// Mitsubishi GX Works2 project: LG WM Press 21.07.21_Conv   PLC: Q03UDV
// LG WM Press 21.07.21_Conv

PROGRAM MAIN
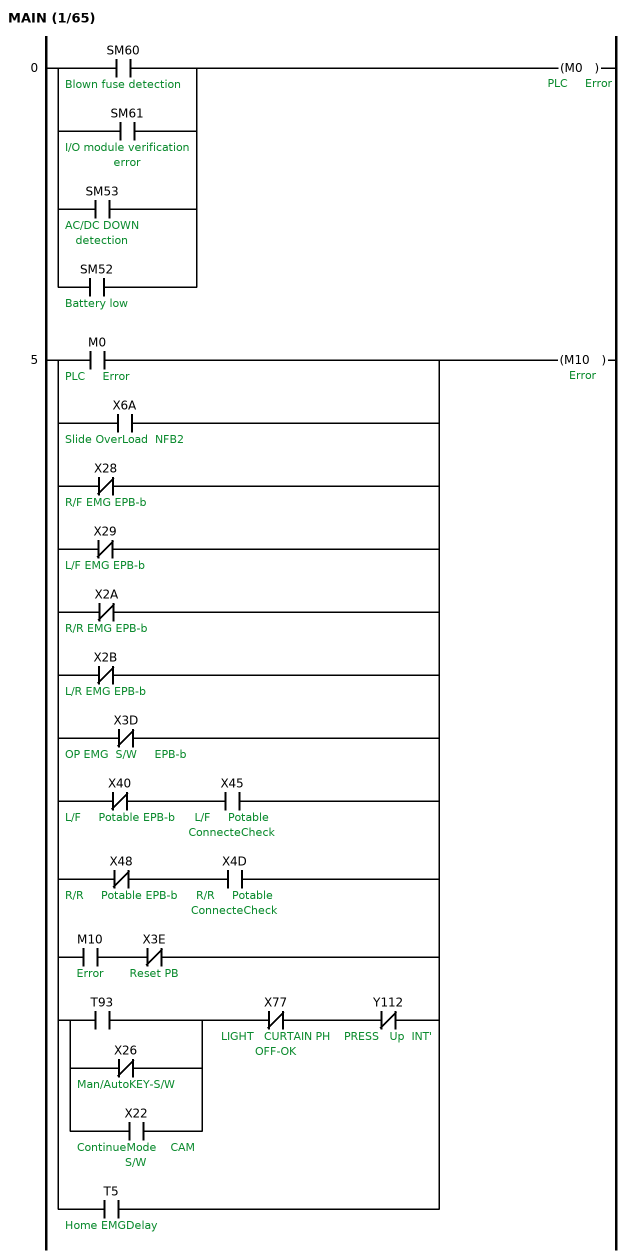
0     LD      SM60  ; Blown fuse detection
      OR      SM61  ; I/O module verification error
      OR      SM53  ; AC/DC DOWN detection
      OR      SM52  ; Battery low
      OUT     M0  ; PLC     Error
5     LD      M0  ; PLC     Error
      OR      X6A  ; Slide OverLoad  NFB2
      ORI     X28  ; R/F EMG EPB-b
      ORI     X29  ; L/F EMG EPB-b
      ORI     X2A  ; R/R EMG EPB-b
      ORI     X2B  ; L/R EMG EPB-b
      ORI     X3D  ; OP EMG  S/W     EPB-b
      LDI     X40  ; L/F     Potable EPB-b
      AND     X45  ; L/F     Potable ConnecteCheck
      ORB
      LDI     X48  ; R/R     Potable EPB-b
      AND     X4D  ; R/R     Potable ConnecteCheck
      ORB
      LD      M10  ; Error
      ANI     X3E  ; Reset PB
      ORB
      LD      T93
      ORI     X26  ; Man/AutoKEY-S/W
      OR      X22  ; ContinueMode    CAM S/W
      ANI     X77  ; LIGHT   CURTAIN PH      OFF-OK
      ANI     Y112  ; PRESS   Up  INT'
      ORB
      OR      T5  ; Home EMGDelay
      OUT     M10  ; Error
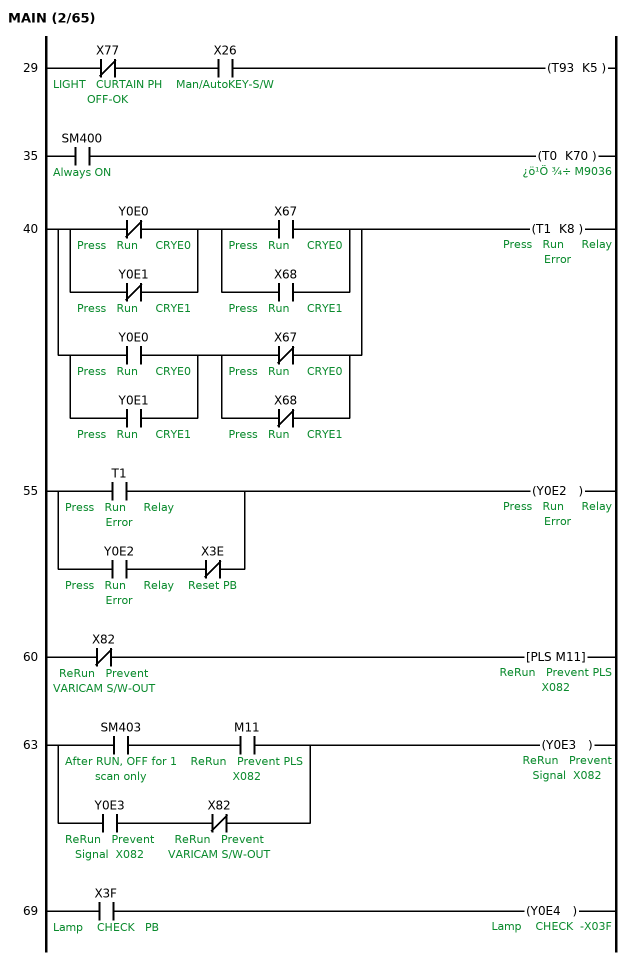
29    LDI     X77  ; LIGHT   CURTAIN PH      OFF-OK
      AND     X26  ; Man/AutoKEY-S/W
      OUT     T93 K5
35    LD      SM400  ; Always ON
      OUT     T0 K70  ; ¿ö¹Ö ¾÷ M9036
40    LDI     Y0E0  ; Press   Run     CRYE0
      ORI     Y0E1  ; Press   Run     CRYE1
      LD      X67  ; Press   Run     CRYE0
      OR      X68  ; Press   Run     CRYE1
      ANB
      LD      Y0E0  ; Press   Run     CRYE0
      OR      Y0E1  ; Press   Run     CRYE1
      LDI     X67  ; Press   Run     CRYE0
      ORI     X68  ; Press   Run     CRYE1
      ANB
      ORB
      OUT     T1 K8  ; Press   Run     Relay   Error
55    LD      T1  ; Press   Run     Relay   Error
      LD      Y0E2  ; Press   Run     Relay   Error
      ANI     X3E  ; Reset PB
      ORB
      OUT     Y0E2  ; Press   Run     Relay   Error
60    LDI     X82  ; ReRun   Prevent VARICAM S/W-OUT
      PLS     M11  ; ReRun   Prevent PLS X082
63    LD      SM403  ; After RUN, OFF for 1 scan only
      AND     M11  ; ReRun   Prevent PLS X082
      LD      Y0E3  ; ReRun   Prevent Signal  X082
      ANI     X82  ; ReRun   Prevent VARICAM S/W-OUT
      ORB
      OUT     Y0E3  ; ReRun   Prevent Signal  X082
69    LD      X3F  ; Lamp    CHECK   PB
      OUT     Y0E4  ; Lamp    CHECK  -X03F
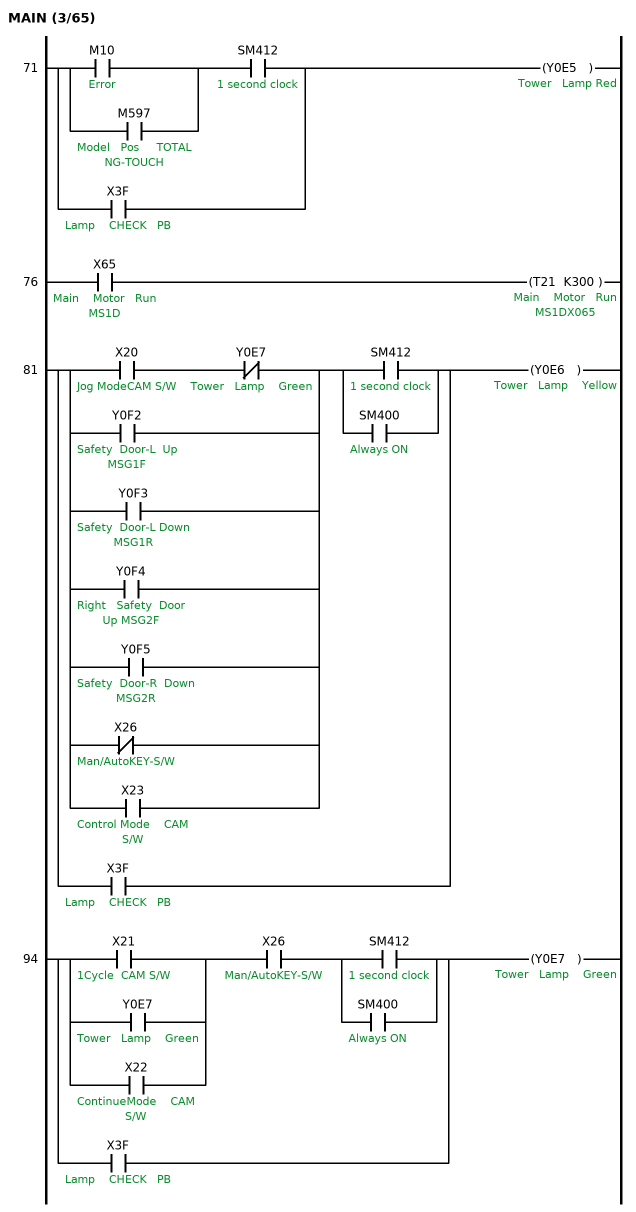
71    LD      M10  ; Error
      OR      M597  ; Model   Pos     TOTAL   NG-TOUCH
      AND     SM412  ; 1 second clock
      OR      X3F  ; Lamp    CHECK   PB
      OUT     Y0E5  ; Tower   Lamp Red
76    LD      X65  ; Main    Motor   Run MS1D
      OUT     T21 K300  ; Main    Motor   Run MS1DX065
81    LD      X20  ; Jog ModeCAM S/W
      ANI     Y0E7  ; Tower   Lamp    Green
      OR      Y0F2  ; Safety  Door-L  Up MSG1F
      OR      Y0F3  ; Safety  Door-L Down     MSG1R
      OR      Y0F4  ; Right   Safety  Door Up MSG2F
      OR      Y0F5  ; Safety  Door-R  Down    MSG2R
      ORI     X26  ; Man/AutoKEY-S/W
      OR      X23  ; Control Mode    CAM S/W
      LD      SM412  ; 1 second clock
      OR      SM400  ; Always ON
      ANB
      OR      X3F  ; Lamp    CHECK   PB
      OUT     Y0E6  ; Tower   Lamp    Yellow
94    LD      X21  ; 1Cycle  CAM S/W
      OR      Y0E7  ; Tower   Lamp    Green
      OR      X22  ; ContinueMode    CAM S/W
      AND     X26  ; Man/AutoKEY-S/W
      LD      SM412  ; 1 second clock
      OR      SM400  ; Always ON
      ANB
      OR      X3F  ; Lamp    CHECK   PB
      OUT     Y0E7  ; Tower   Lamp    Green
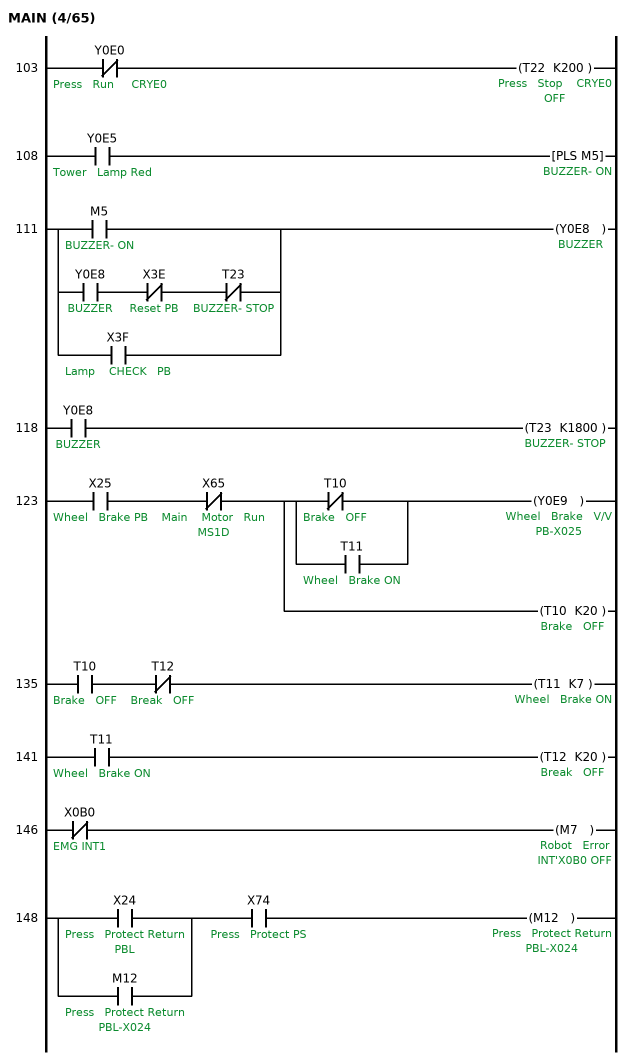
103   LDI     Y0E0  ; Press   Run     CRYE0
      OUT     T22 K200  ; Press   Stop    CRYE0   OFF
108   LD      Y0E5  ; Tower   Lamp Red
      PLS     M5  ; BUZZER- ON
111   LD      M5  ; BUZZER- ON
      LD      Y0E8  ; BUZZER
      ANI     X3E  ; Reset PB
      ANI     T23  ; BUZZER- STOP
      ORB
      OR      X3F  ; Lamp    CHECK   PB
      OUT     Y0E8  ; BUZZER
118   LD      Y0E8  ; BUZZER
      OUT     T23 K1800  ; BUZZER- STOP
123   LD      X25  ; Wheel   Brake PB
      ANI     X65  ; Main    Motor   Run MS1D
      MPS
      LDI     T10  ; Brake   OFF
      OR      T11  ; Wheel   Brake ON
      ANB
      OUT     Y0E9  ; Wheel   Brake   V/V     PB-X025
      MPP
      OUT     T10 K20  ; Brake   OFF
135   LD      T10  ; Brake   OFF
      ANI     T12  ; Break   OFF
      OUT     T11 K7  ; Wheel   Brake ON
141   LD      T11  ; Wheel   Brake ON
      OUT     T12 K20  ; Break   OFF
146   LDI     X0B0  ; EMG INT1
      OUT     M7  ; Robot   Error   INT'X0B0 OFF
148   LD      X24  ; Press   Protect Return  PBL
      OR      M12  ; Press   Protect Return  PBL-X024
      AND     X74  ; Press   Protect PS
      OUT     M12  ; Press   Protect Return  PBL-X024
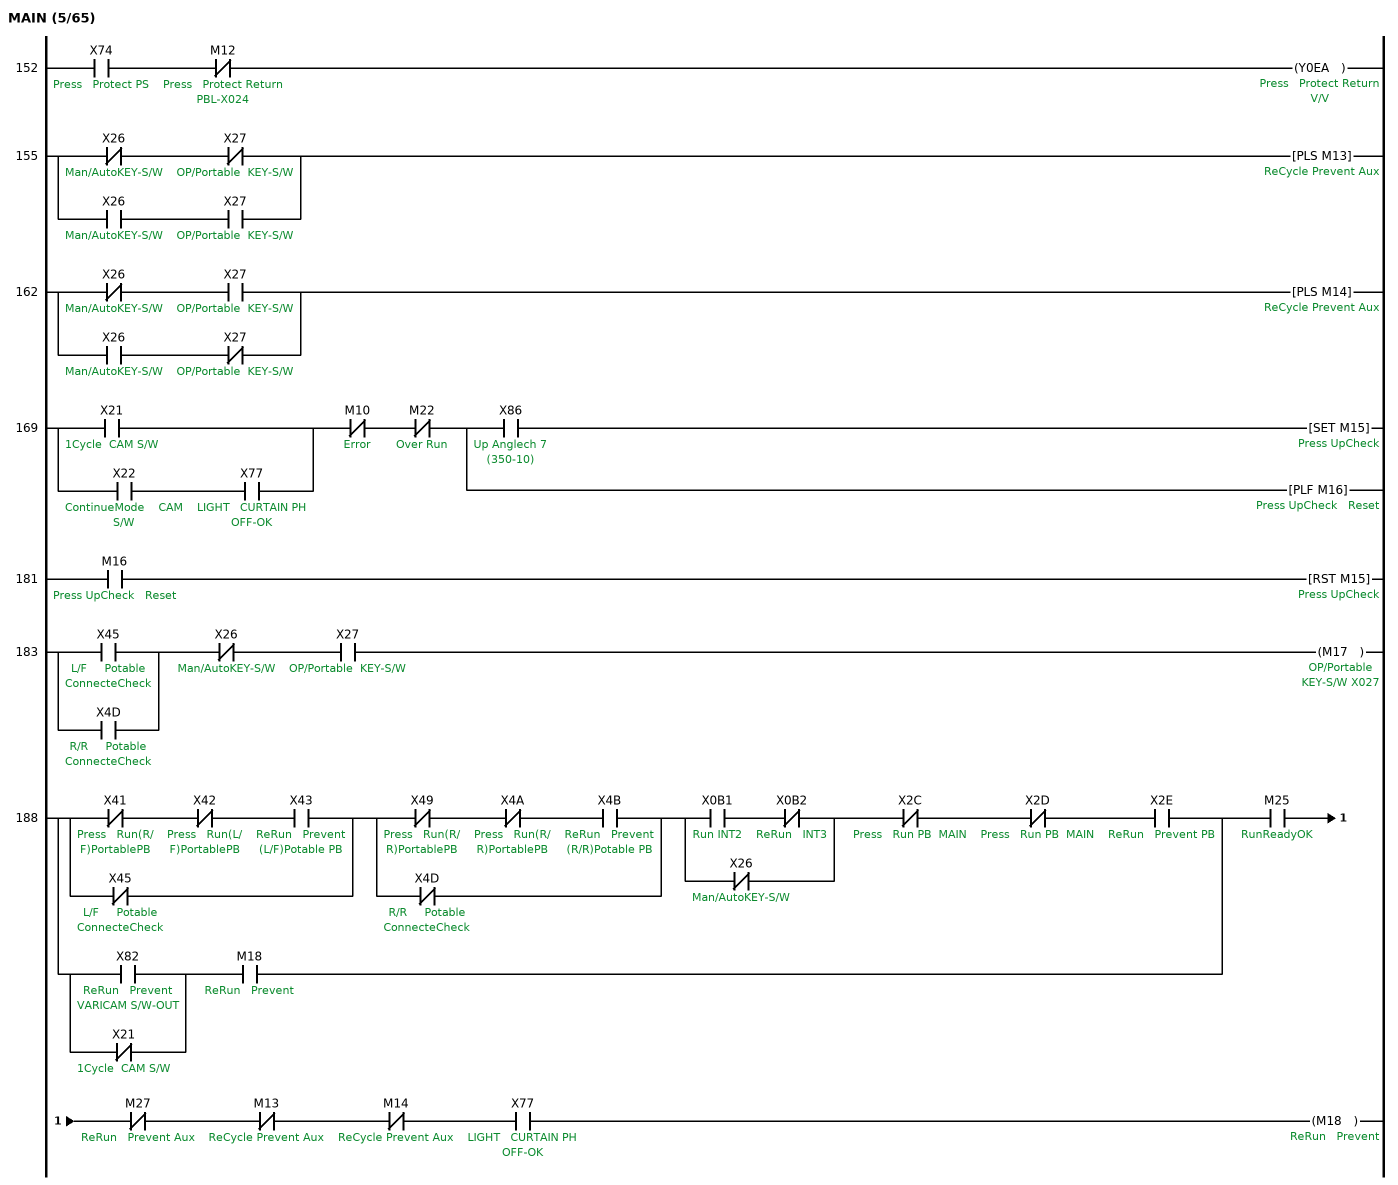
152   LD      X74  ; Press   Protect PS
      ANI     M12  ; Press   Protect Return  PBL-X024
      OUT     Y0EA  ; Press   Protect Return  V/V
155   LDI     X26  ; Man/AutoKEY-S/W
      ANI     X27  ; OP/Portable  KEY-S/W
      LD      X26  ; Man/AutoKEY-S/W
      AND     X27  ; OP/Portable  KEY-S/W
      ORB
      PLS     M13  ; ReCycle Prevent Aux
162   LDI     X26  ; Man/AutoKEY-S/W
      AND     X27  ; OP/Portable  KEY-S/W
      LD      X26  ; Man/AutoKEY-S/W
      ANI     X27  ; OP/Portable  KEY-S/W
      ORB
      PLS     M14  ; ReCycle Prevent Aux
169   LD      X21  ; 1Cycle  CAM S/W
      LD      X22  ; ContinueMode    CAM S/W
      AND     X77  ; LIGHT   CURTAIN PH      OFF-OK
      ORB
      ANI     M10  ; Error
      ANI     M22  ; Over Run
      MPS
      AND     X86  ; Up Anglech 7    (350-10)
      SET     M15  ; Press UpCheck
      MPP
      PLF     M16  ; Press UpCheck   Reset
181   LD      M16  ; Press UpCheck   Reset
      RST     M15  ; Press UpCheck
183   LD      X45  ; L/F     Potable ConnecteCheck
      OR      X4D  ; R/R     Potable ConnecteCheck
      ANI     X26  ; Man/AutoKEY-S/W
      AND     X27  ; OP/Portable  KEY-S/W
      OUT     M17  ; OP/Portable     KEY-S/W X027
188   LDI     X41  ; Press   Run(R/F)PortablePB
      ANI     X42  ; Press   Run(L/F)PortablePB
      AND     X43  ; ReRun   Prevent (L/F)Potable PB
      ORI     X45  ; L/F     Potable ConnecteCheck
      LDI     X49  ; Press   Run(R/R)PortablePB
      ANI     X4A  ; Press   Run(R/R)PortablePB
      AND     X4B  ; ReRun   Prevent (R/R)Potable PB
      ORI     X4D  ; R/R     Potable ConnecteCheck
      ANB
      LD      X0B1  ; Run INT2
      ANI     X0B2  ; ReRun   INT3
      ORI     X26  ; Man/AutoKEY-S/W
      ANB
      ANI     X2C  ; Press   Run PB  MAIN
      ANI     X2D  ; Press   Run PB  MAIN
      AND     X2E  ; ReRun   Prevent PB
      LD      X82  ; ReRun   Prevent VARICAM S/W-OUT
      ORI     X21  ; 1Cycle  CAM S/W
      AND     M18  ; ReRun   Prevent
      ORB
      AND     M25  ; RunReadyOK
      ANI     M27  ; ReRun   Prevent Aux
      ANI     M13  ; ReCycle Prevent Aux
      ANI     M14  ; ReCycle Prevent Aux
      AND     X77  ; LIGHT   CURTAIN PH      OFF-OK
      OUT     M18  ; ReRun   Prevent
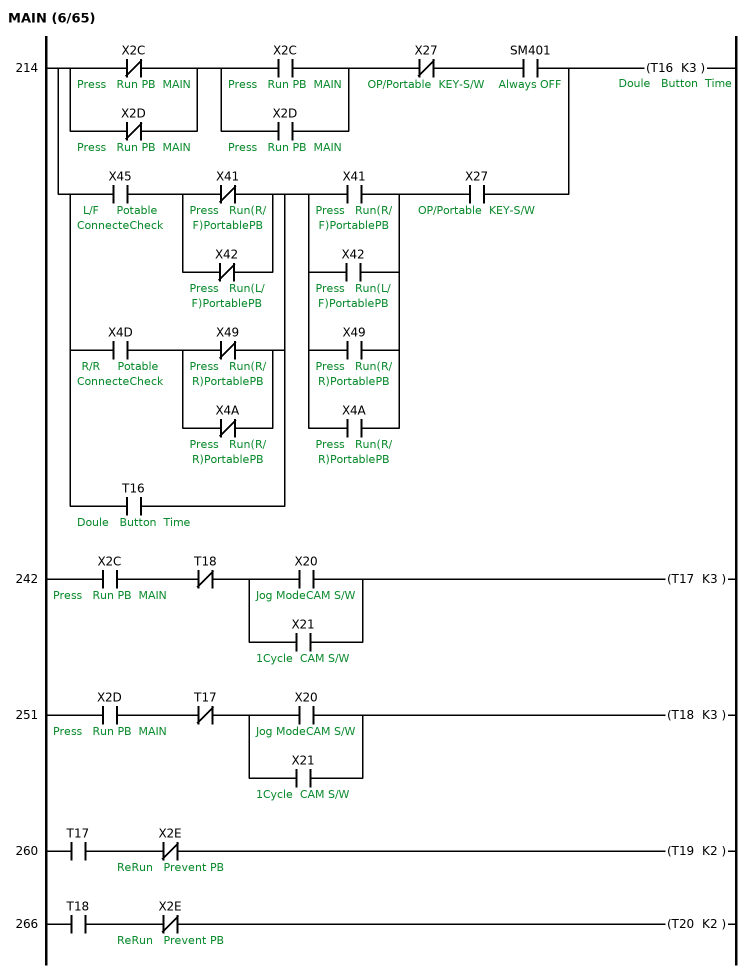
214   LDI     X2C  ; Press   Run PB  MAIN
      ORI     X2D  ; Press   Run PB  MAIN
      LD      X2C  ; Press   Run PB  MAIN
      OR      X2D  ; Press   Run PB  MAIN
      ANB
      ANI     X27  ; OP/Portable  KEY-S/W
      AND     SM401  ; Always OFF
      LD      X45  ; L/F     Potable ConnecteCheck
      LDI     X41  ; Press   Run(R/F)PortablePB
      ORI     X42  ; Press   Run(L/F)PortablePB
      ANB
      LD      X4D  ; R/R     Potable ConnecteCheck
      LDI     X49  ; Press   Run(R/R)PortablePB
      ORI     X4A  ; Press   Run(R/R)PortablePB
      ANB
      ORB
      OR      T16  ; Doule   Button  Time
      LD      X41  ; Press   Run(R/F)PortablePB
      OR      X42  ; Press   Run(L/F)PortablePB
      OR      X49  ; Press   Run(R/R)PortablePB
      OR      X4A  ; Press   Run(R/R)PortablePB
      ANB
      AND     X27  ; OP/Portable  KEY-S/W
      ORB
      OUT     T16 K3  ; Doule   Button  Time
242   LD      X2C  ; Press   Run PB  MAIN
      ANI     T18
      LD      X20  ; Jog ModeCAM S/W
      OR      X21  ; 1Cycle  CAM S/W
      ANB
      OUT     T17 K3
251   LD      X2D  ; Press   Run PB  MAIN
      ANI     T17
      LD      X20  ; Jog ModeCAM S/W
      OR      X21  ; 1Cycle  CAM S/W
      ANB
      OUT     T18 K3
260   LD      T17
      ANI     X2E  ; ReRun   Prevent PB
      OUT     T19 K2
266   LD      T18
      ANI     X2E  ; ReRun   Prevent PB
      OUT     T20 K2
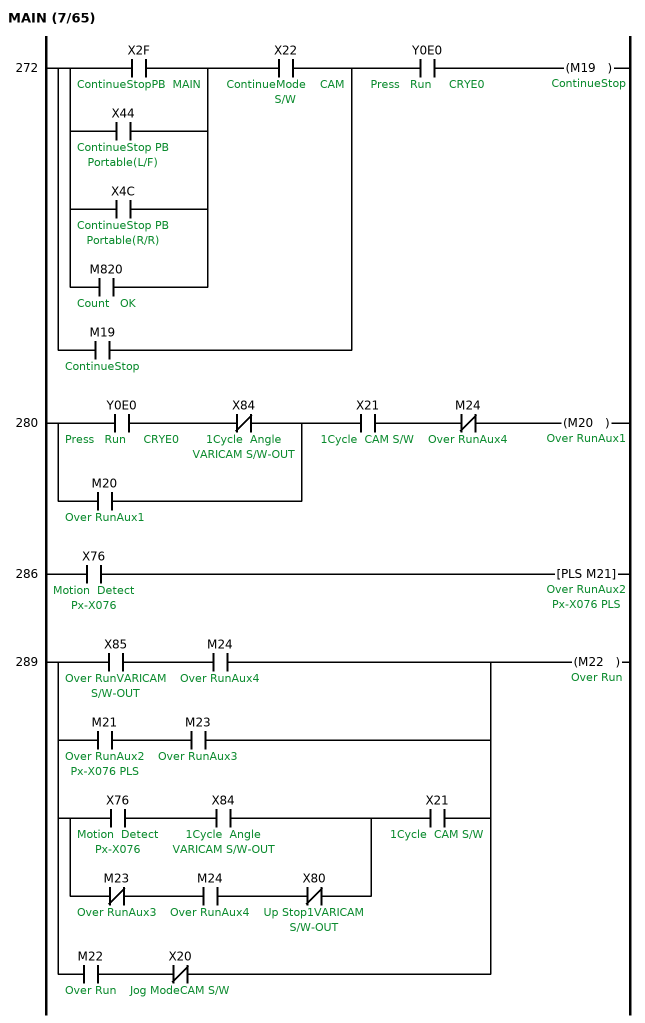
272   LD      X2F  ; ContinueStopPB  MAIN
      OR      X44  ; ContinueStop PB Portable(L/F)
      OR      X4C  ; ContinueStop PB Portable(R/R)
      OR      M820  ; Count   OK
      AND     X22  ; ContinueMode    CAM S/W
      OR      M19  ; ContinueStop
      AND     Y0E0  ; Press   Run     CRYE0
      OUT     M19  ; ContinueStop
280   LD      Y0E0  ; Press   Run     CRYE0
      ANI     X84  ; 1Cycle  Angle   VARICAM S/W-OUT
      OR      M20  ; Over RunAux1
      AND     X21  ; 1Cycle  CAM S/W
      ANI     M24  ; Over RunAux4
      OUT     M20  ; Over RunAux1
286   LD      X76  ; Motion  Detect  Px-X076
      PLS     M21  ; Over RunAux2    Px-X076 PLS
289   LD      X85  ; Over RunVARICAM S/W-OUT
      AND     M24  ; Over RunAux4
      LD      M21  ; Over RunAux2    Px-X076 PLS
      AND     M23  ; Over RunAux3
      ORB
      LD      X76  ; Motion  Detect  Px-X076
      AND     X84  ; 1Cycle  Angle   VARICAM S/W-OUT
      LDI     M23  ; Over RunAux3
      AND     M24  ; Over RunAux4
      ANI     X80  ; Up Stop1VARICAM S/W-OUT
      ORB
      AND     X21  ; 1Cycle  CAM S/W
      ORB
      LD      M22  ; Over Run
      ANI     X20  ; Jog ModeCAM S/W
      ORB
      OUT     M22  ; Over Run
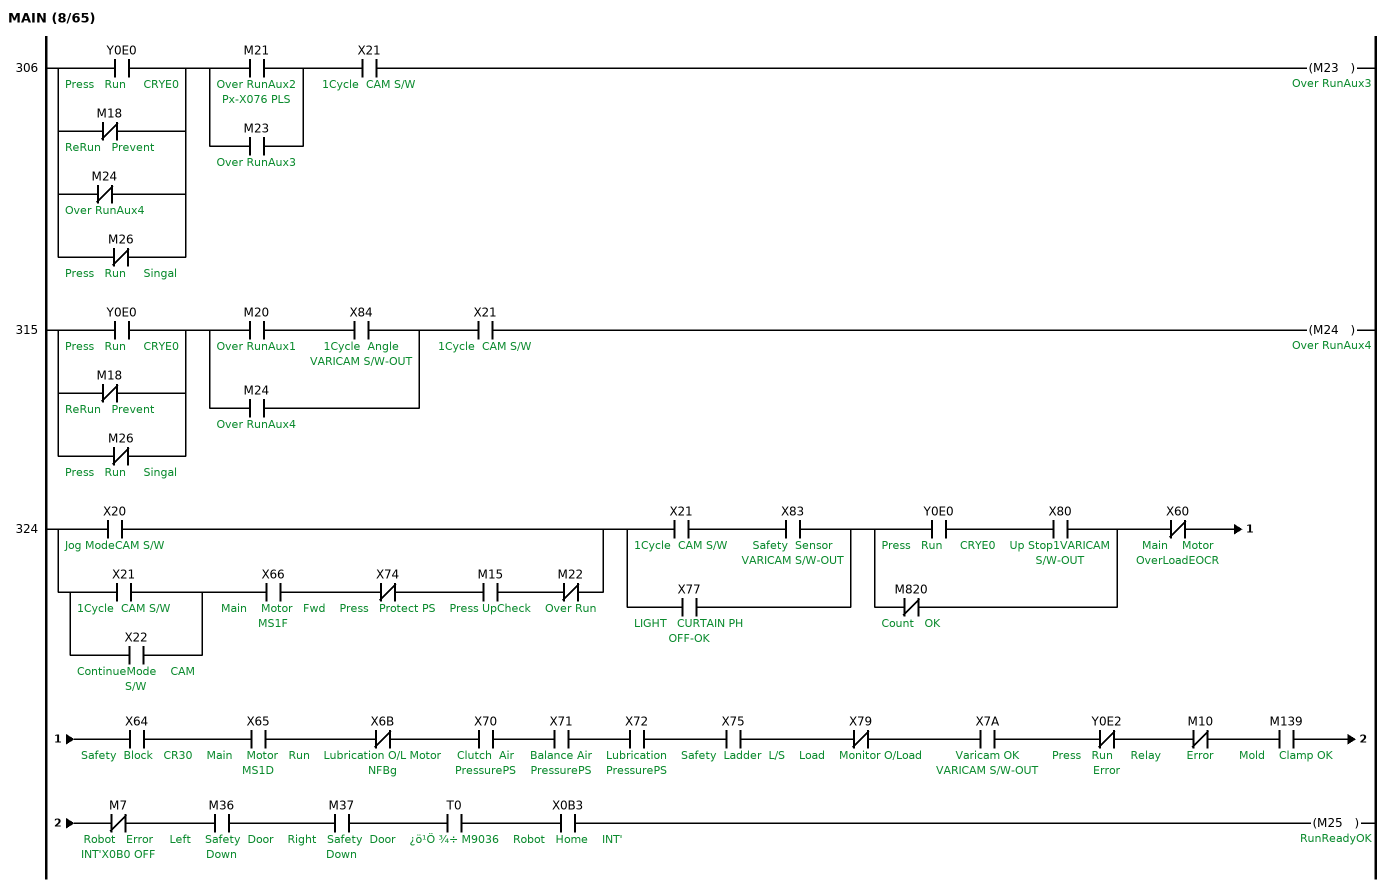
306   LD      Y0E0  ; Press   Run     CRYE0
      ORI     M18  ; ReRun   Prevent
      ORI     M24  ; Over RunAux4
      ORI     M26  ; Press   Run     Singal
      LD      M21  ; Over RunAux2    Px-X076 PLS
      OR      M23  ; Over RunAux3
      ANB
      AND     X21  ; 1Cycle  CAM S/W
      OUT     M23  ; Over RunAux3
315   LD      Y0E0  ; Press   Run     CRYE0
      ORI     M18  ; ReRun   Prevent
      ORI     M26  ; Press   Run     Singal
      LD      M20  ; Over RunAux1
      AND     X84  ; 1Cycle  Angle   VARICAM S/W-OUT
      OR      M24  ; Over RunAux4
      ANB
      AND     X21  ; 1Cycle  CAM S/W
      OUT     M24  ; Over RunAux4
324   LD      X20  ; Jog ModeCAM S/W
      LD      X21  ; 1Cycle  CAM S/W
      OR      X22  ; ContinueMode    CAM S/W
      AND     X66  ; Main    Motor   Fwd     MS1F
      ANI     X74  ; Press   Protect PS
      AND     M15  ; Press UpCheck
      ANI     M22  ; Over Run
      ORB
      LD      X21  ; 1Cycle  CAM S/W
      AND     X83  ; Safety  Sensor  VARICAM S/W-OUT
      OR      X77  ; LIGHT   CURTAIN PH      OFF-OK
      ANB
      LD      Y0E0  ; Press   Run     CRYE0
      AND     X80  ; Up Stop1VARICAM S/W-OUT
      ORI     M820  ; Count   OK
      ANB
      ANI     X60  ; Main    Motor   OverLoadEOCR
      AND     X64  ; Safety  Block   CR30
      AND     X65  ; Main    Motor   Run MS1D
      ANI     X6B  ; Lubrication O/L Motor   NFBg
      AND     X70  ; Clutch  Air     PressurePS
      AND     X71  ; Balance Air     PressurePS
      AND     X72  ; Lubrication     PressurePS
      AND     X75  ; Safety  Ladder  L/S
      ANI     X79  ; Load    Monitor O/Load
      AND     X7A  ; Varicam OK      VARICAM S/W-OUT
      ANI     Y0E2  ; Press   Run     Relay   Error
      ANI     M10  ; Error
      AND     M139  ; Mold    Clamp OK
      ANI     M7  ; Robot   Error   INT'X0B0 OFF
      AND     M36  ; Left    Safety  Door    Down
      AND     M37  ; Right   Safety  Door    Down
      AND     T0  ; ¿ö¹Ö ¾÷ M9036
      AND     X0B3  ; Robot   Home    INT'
      OUT     M25  ; RunReadyOK
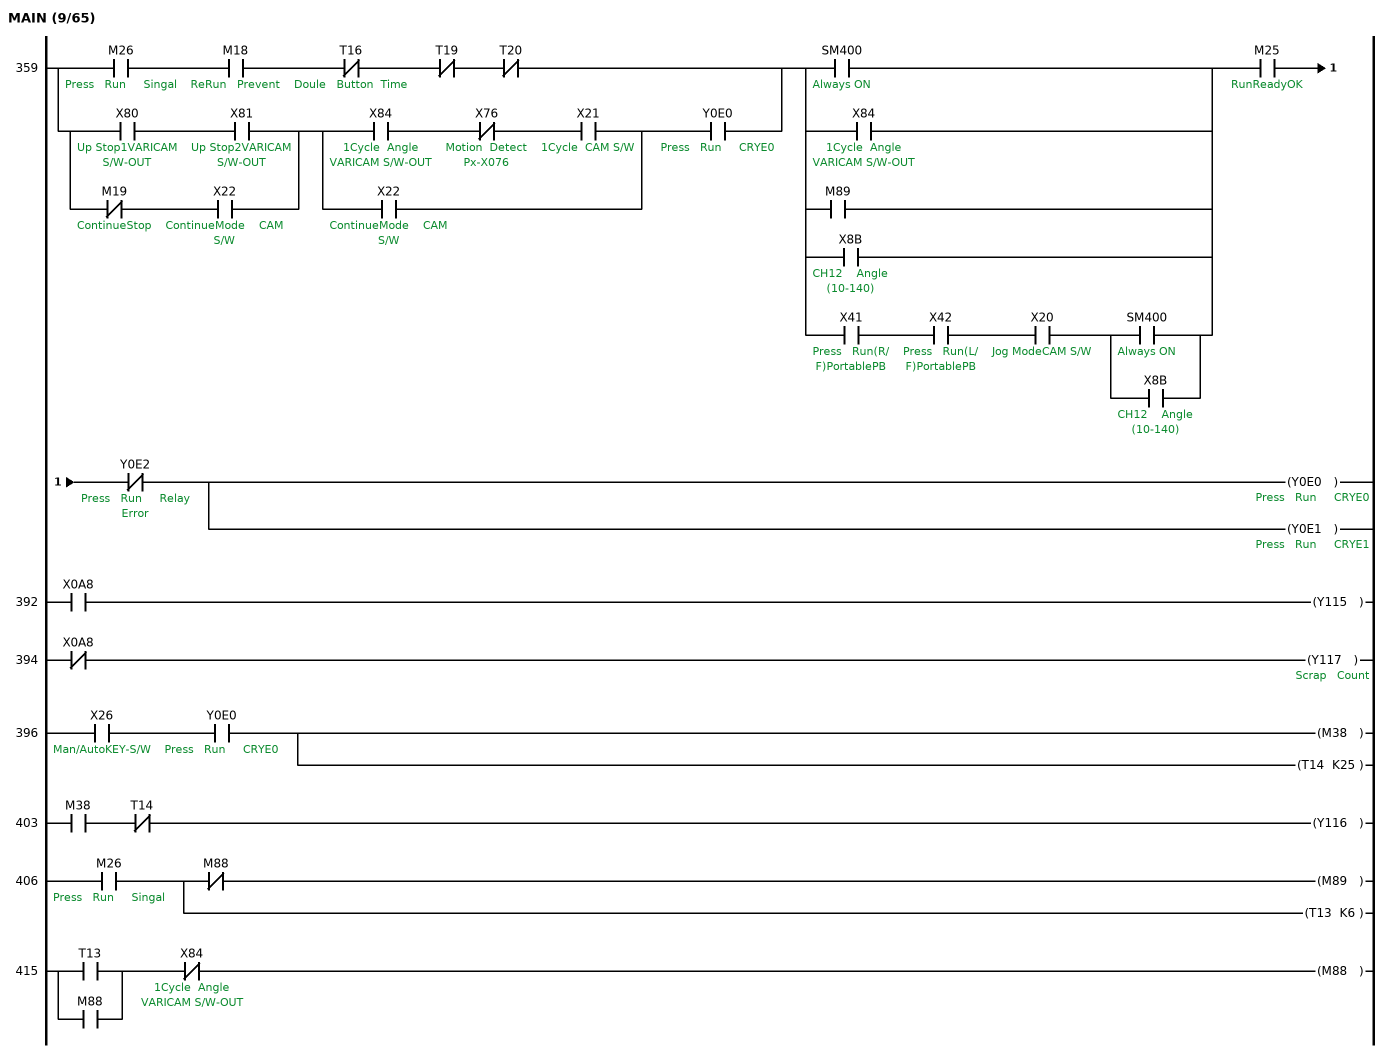
359   LD      M26  ; Press   Run     Singal
      AND     M18  ; ReRun   Prevent
      ANI     T16  ; Doule   Button  Time
      ANI     T19
      ANI     T20
      LD      X80  ; Up Stop1VARICAM S/W-OUT
      AND     X81  ; Up Stop2VARICAM S/W-OUT
      LDI     M19  ; ContinueStop
      AND     X22  ; ContinueMode    CAM S/W
      ORB
      LD      X84  ; 1Cycle  Angle   VARICAM S/W-OUT
      ANI     X76  ; Motion  Detect  Px-X076
      AND     X21  ; 1Cycle  CAM S/W
      OR      X22  ; ContinueMode    CAM S/W
      ANB
      AND     Y0E0  ; Press   Run     CRYE0
      ORB
      LD      SM400  ; Always ON
      OR      X84  ; 1Cycle  Angle   VARICAM S/W-OUT
      OR      M89
      OR      X8B  ; CH12    Angle   (10-140)
      LD      X41  ; Press   Run(R/F)PortablePB
      AND     X42  ; Press   Run(L/F)PortablePB
      AND     X20  ; Jog ModeCAM S/W
      LD      SM400  ; Always ON
      OR      X8B  ; CH12    Angle   (10-140)
      ANB
      ORB
      ANB
      AND     M25  ; RunReadyOK
      ANI     Y0E2  ; Press   Run     Relay   Error
      OUT     Y0E0  ; Press   Run     CRYE0
      OUT     Y0E1  ; Press   Run     CRYE1
392   LD      X0A8
      OUT     Y115
394   LDI     X0A8
      OUT     Y117  ; Scrap   Count
396   LD      X26  ; Man/AutoKEY-S/W
      AND     Y0E0  ; Press   Run     CRYE0
      OUT     M38
      OUT     T14 K25
403   LD      M38
      ANI     T14
      OUT     Y116
406   LD      M26  ; Press   Run     Singal
      MPS
      ANI     M88
      OUT     M89
      MPP
      OUT     T13 K6
415   LD      T13
      OR      M88
      ANI     X84  ; 1Cycle  Angle   VARICAM S/W-OUT
      OUT     M88
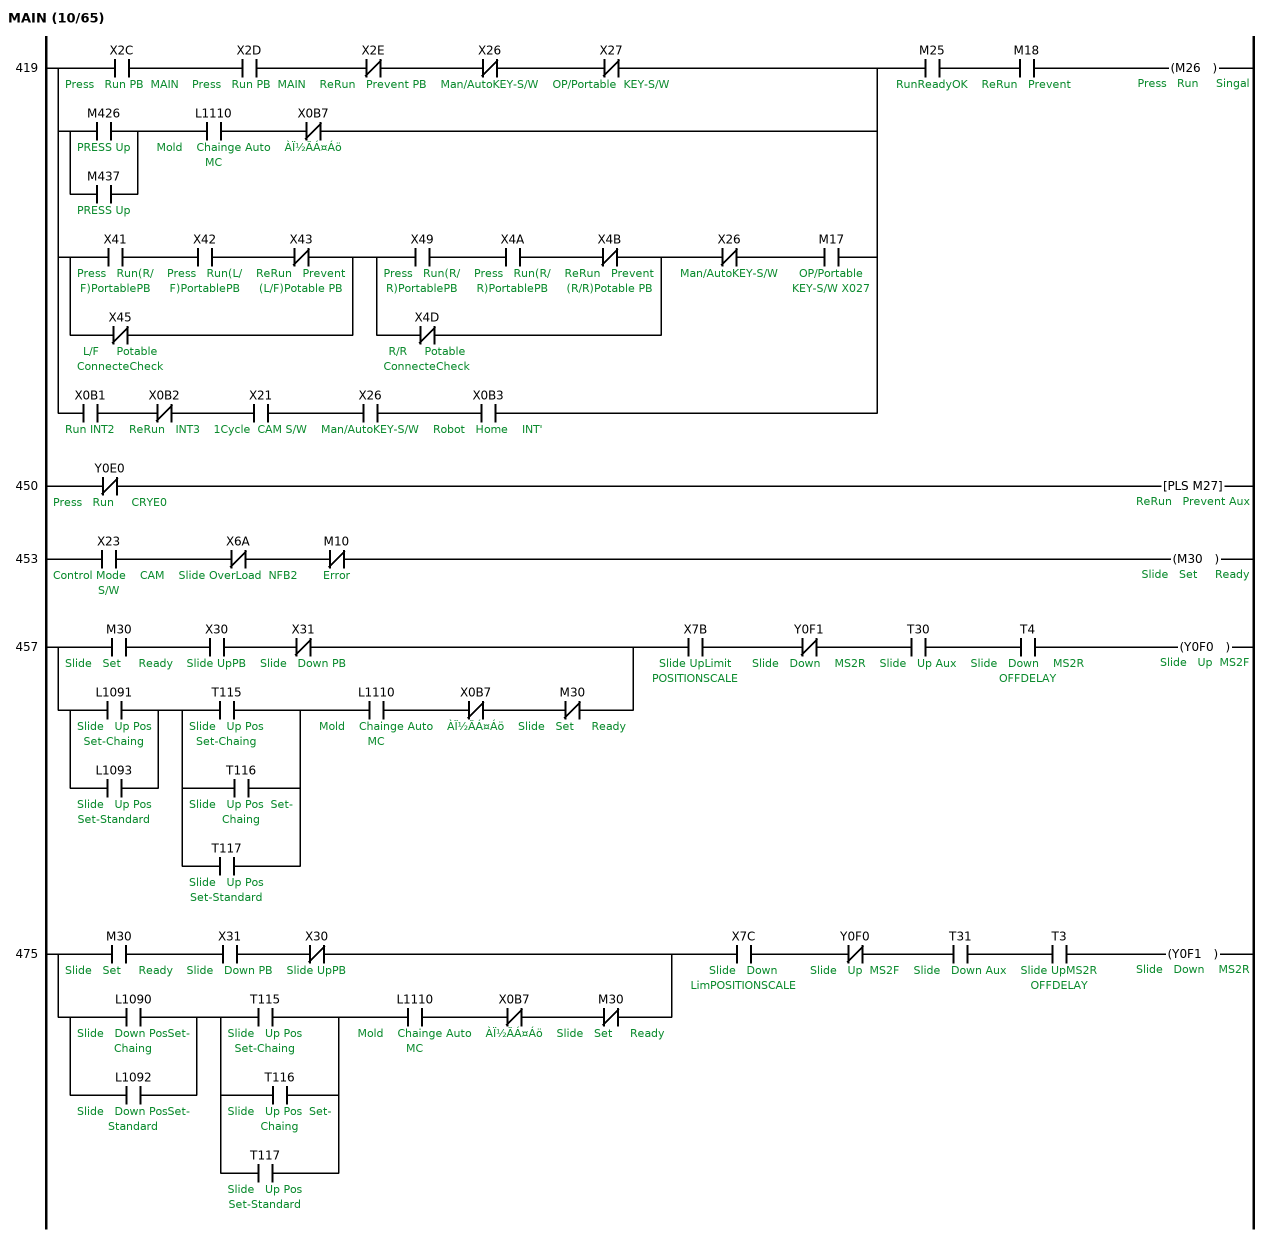
419   LD      X2C  ; Press   Run PB  MAIN
      AND     X2D  ; Press   Run PB  MAIN
      ANI     X2E  ; ReRun   Prevent PB
      ANI     X26  ; Man/AutoKEY-S/W
      ANI     X27  ; OP/Portable  KEY-S/W
      LD      M426  ; PRESS Up
      OR      M437  ; PRESS Up
      AND     L1110  ; Mold    Chainge Auto MC
      ANI     X0B7  ; ÀÏ½ÃÁ¤Áö
      ORB
      LD      X41  ; Press   Run(R/F)PortablePB
      AND     X42  ; Press   Run(L/F)PortablePB
      ANI     X43  ; ReRun   Prevent (L/F)Potable PB
      ORI     X45  ; L/F     Potable ConnecteCheck
      LD      X49  ; Press   Run(R/R)PortablePB
      AND     X4A  ; Press   Run(R/R)PortablePB
      ANI     X4B  ; ReRun   Prevent (R/R)Potable PB
      ORI     X4D  ; R/R     Potable ConnecteCheck
      ANB
      ANI     X26  ; Man/AutoKEY-S/W
      AND     M17  ; OP/Portable     KEY-S/W X027
      ORB
      LD      X0B1  ; Run INT2
      ANI     X0B2  ; ReRun   INT3
      AND     X21  ; 1Cycle  CAM S/W
      AND     X26  ; Man/AutoKEY-S/W
      AND     X0B3  ; Robot   Home    INT'
      ORB
      AND     M25  ; RunReadyOK
      AND     M18  ; ReRun   Prevent
      OUT     M26  ; Press   Run     Singal
450   LDI     Y0E0  ; Press   Run     CRYE0
      PLS     M27  ; ReRun   Prevent Aux
453   LD      X23  ; Control Mode    CAM S/W
      ANI     X6A  ; Slide OverLoad  NFB2
      ANI     M10  ; Error
      OUT     M30  ; Slide   Set     Ready
457   LD      M30  ; Slide   Set     Ready
      AND     X30  ; Slide UpPB
      ANI     X31  ; Slide   Down PB
      LD      L1091  ; Slide   Up Pos  Set-Chaing
      OR      L1093  ; Slide   Up Pos  Set-Standard
      LD      T115  ; Slide   Up Pos  Set-Chaing
      OR      T116  ; Slide   Up Pos  Set-    Chaing
      OR      T117  ; Slide   Up Pos  Set-Standard
      ANB
      AND     L1110  ; Mold    Chainge Auto MC
      ANI     X0B7  ; ÀÏ½ÃÁ¤Áö
      ANI     M30  ; Slide   Set     Ready
      ORB
      AND     X7B  ; Slide UpLimit   POSITIONSCALE
      ANI     Y0F1  ; Slide   Down    MS2R
      AND     T30  ; Slide   Up Aux
      AND     T4  ; Slide   Down    MS2R OFFDELAY
      OUT     Y0F0  ; Slide   Up  MS2F
475   LD      M30  ; Slide   Set     Ready
      AND     X31  ; Slide   Down PB
      ANI     X30  ; Slide UpPB
      LD      L1090  ; Slide   Down PosSet-    Chaing
      OR      L1092  ; Slide   Down PosSet-    Standard
      LD      T115  ; Slide   Up Pos  Set-Chaing
      OR      T116  ; Slide   Up Pos  Set-    Chaing
      OR      T117  ; Slide   Up Pos  Set-Standard
      ANB
      AND     L1110  ; Mold    Chainge Auto MC
      ANI     X0B7  ; ÀÏ½ÃÁ¤Áö
      ANI     M30  ; Slide   Set     Ready
      ORB
      AND     X7C  ; Slide   Down LimPOSITIONSCALE
      ANI     Y0F0  ; Slide   Up  MS2F
      AND     T31  ; Slide   Down Aux
      AND     T3  ; Slide UpMS2R OFFDELAY
      OUT     Y0F1  ; Slide   Down    MS2R
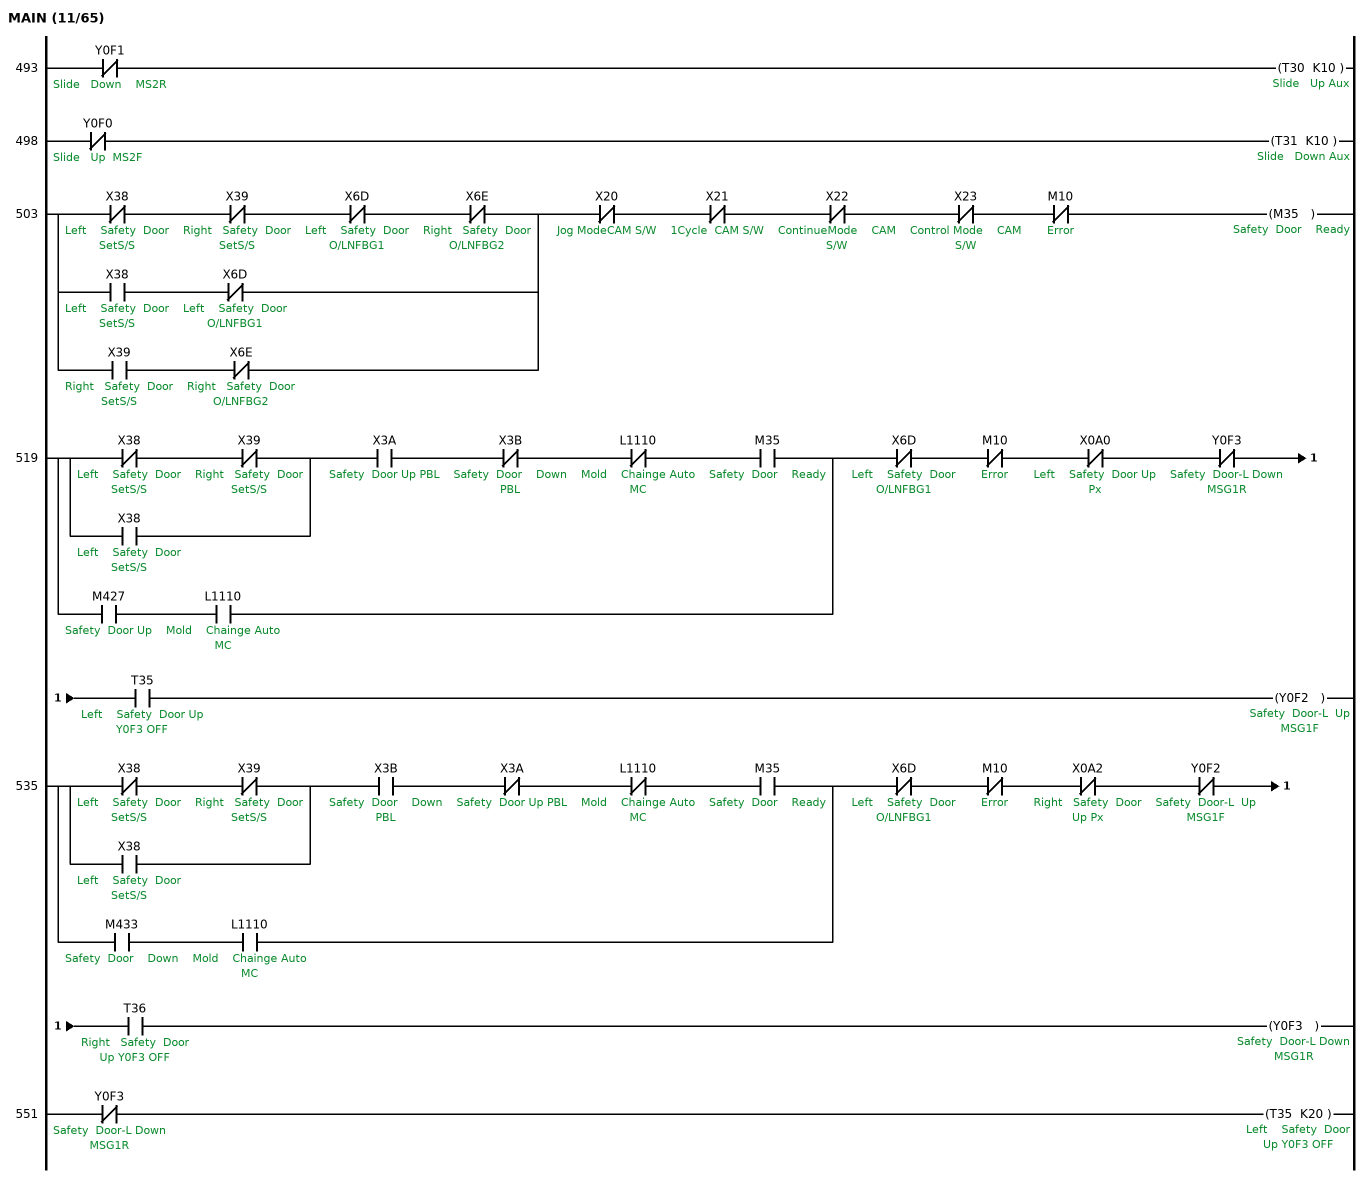
493   LDI     Y0F1  ; Slide   Down    MS2R
      OUT     T30 K10  ; Slide   Up Aux
498   LDI     Y0F0  ; Slide   Up  MS2F
      OUT     T31 K10  ; Slide   Down Aux
503   LDI     X38  ; Left    Safety  Door SetS/S
      ANI     X39  ; Right   Safety  Door SetS/S
      ANI     X6D  ; Left    Safety  Door O/LNFBG1
      ANI     X6E  ; Right   Safety  Door O/LNFBG2
      LD      X38  ; Left    Safety  Door SetS/S
      ANI     X6D  ; Left    Safety  Door O/LNFBG1
      ORB
      LD      X39  ; Right   Safety  Door SetS/S
      ANI     X6E  ; Right   Safety  Door O/LNFBG2
      ORB
      ANI     X20  ; Jog ModeCAM S/W
      ANI     X21  ; 1Cycle  CAM S/W
      ANI     X22  ; ContinueMode    CAM S/W
      ANI     X23  ; Control Mode    CAM S/W
      ANI     M10  ; Error
      OUT     M35  ; Safety  Door    Ready
519   LDI     X38  ; Left    Safety  Door SetS/S
      ANI     X39  ; Right   Safety  Door SetS/S
      OR      X38  ; Left    Safety  Door SetS/S
      AND     X3A  ; Safety  Door Up PBL
      ANI     X3B  ; Safety  Door    Down PBL
      ANI     L1110  ; Mold    Chainge Auto MC
      AND     M35  ; Safety  Door    Ready
      LD      M427  ; Safety  Door Up
      AND     L1110  ; Mold    Chainge Auto MC
      ORB
      ANI     X6D  ; Left    Safety  Door O/LNFBG1
      ANI     M10  ; Error
      ANI     X0A0  ; Left    Safety  Door Up Px
      ANI     Y0F3  ; Safety  Door-L Down     MSG1R
      AND     T35  ; Left    Safety  Door Up Y0F3 OFF
      OUT     Y0F2  ; Safety  Door-L  Up MSG1F
535   LDI     X38  ; Left    Safety  Door SetS/S
      ANI     X39  ; Right   Safety  Door SetS/S
      OR      X38  ; Left    Safety  Door SetS/S
      AND     X3B  ; Safety  Door    Down PBL
      ANI     X3A  ; Safety  Door Up PBL
      ANI     L1110  ; Mold    Chainge Auto MC
      AND     M35  ; Safety  Door    Ready
      LD      M433  ; Safety  Door    Down
      AND     L1110  ; Mold    Chainge Auto MC
      ORB
      ANI     X6D  ; Left    Safety  Door O/LNFBG1
      ANI     M10  ; Error
      ANI     X0A2  ; Right   Safety  Door Up Px
      ANI     Y0F2  ; Safety  Door-L  Up MSG1F
      AND     T36  ; Right   Safety  Door Up Y0F3 OFF
      OUT     Y0F3  ; Safety  Door-L Down     MSG1R
551   LDI     Y0F3  ; Safety  Door-L Down     MSG1R
      OUT     T35 K20  ; Left    Safety  Door Up Y0F3 OFF
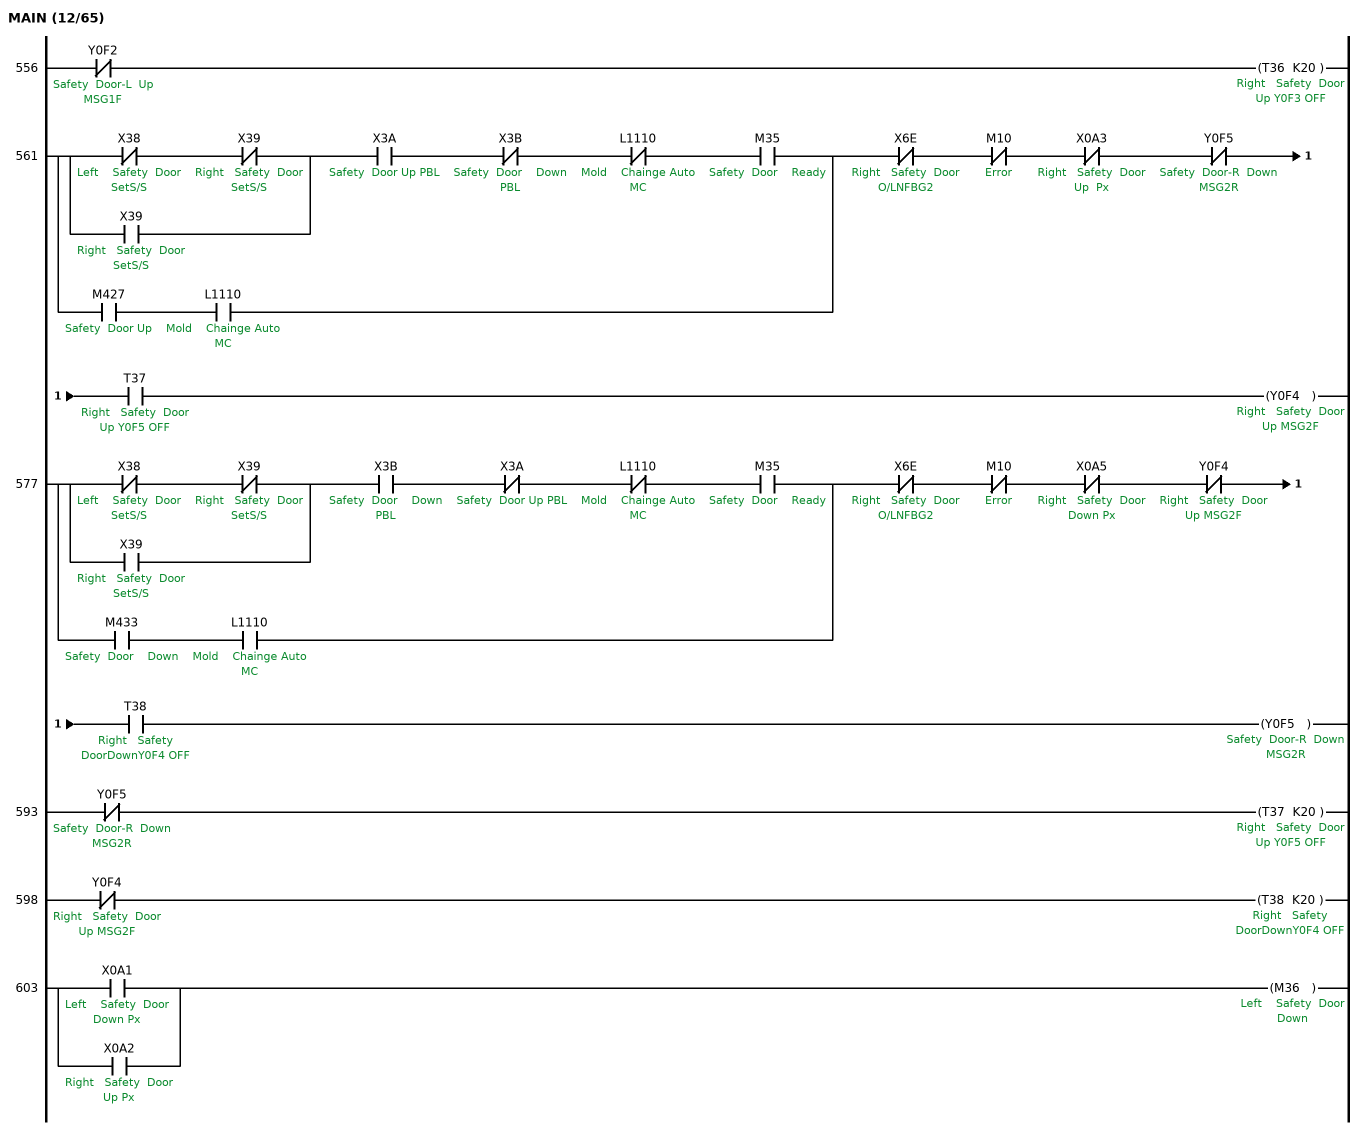
556   LDI     Y0F2  ; Safety  Door-L  Up MSG1F
      OUT     T36 K20  ; Right   Safety  Door Up Y0F3 OFF
561   LDI     X38  ; Left    Safety  Door SetS/S
      ANI     X39  ; Right   Safety  Door SetS/S
      OR      X39  ; Right   Safety  Door SetS/S
      AND     X3A  ; Safety  Door Up PBL
      ANI     X3B  ; Safety  Door    Down PBL
      ANI     L1110  ; Mold    Chainge Auto MC
      AND     M35  ; Safety  Door    Ready
      LD      M427  ; Safety  Door Up
      AND     L1110  ; Mold    Chainge Auto MC
      ORB
      ANI     X6E  ; Right   Safety  Door O/LNFBG2
      ANI     M10  ; Error
      ANI     X0A3  ; Right   Safety  Door Up  Px
      ANI     Y0F5  ; Safety  Door-R  Down    MSG2R
      AND     T37  ; Right   Safety  Door Up Y0F5 OFF
      OUT     Y0F4  ; Right   Safety  Door Up MSG2F
577   LDI     X38  ; Left    Safety  Door SetS/S
      ANI     X39  ; Right   Safety  Door SetS/S
      OR      X39  ; Right   Safety  Door SetS/S
      AND     X3B  ; Safety  Door    Down PBL
      ANI     X3A  ; Safety  Door Up PBL
      ANI     L1110  ; Mold    Chainge Auto MC
      AND     M35  ; Safety  Door    Ready
      LD      M433  ; Safety  Door    Down
      AND     L1110  ; Mold    Chainge Auto MC
      ORB
      ANI     X6E  ; Right   Safety  Door O/LNFBG2
      ANI     M10  ; Error
      ANI     X0A5  ; Right   Safety  Door    Down Px
      ANI     Y0F4  ; Right   Safety  Door Up MSG2F
      AND     T38  ; Right   Safety  DoorDownY0F4 OFF
      OUT     Y0F5  ; Safety  Door-R  Down    MSG2R
593   LDI     Y0F5  ; Safety  Door-R  Down    MSG2R
      OUT     T37 K20  ; Right   Safety  Door Up Y0F5 OFF
598   LDI     Y0F4  ; Right   Safety  Door Up MSG2F
      OUT     T38 K20  ; Right   Safety  DoorDownY0F4 OFF
603   LD      X0A1  ; Left    Safety  Door    Down Px
      OR      X0A2  ; Right   Safety  Door Up Px
      OUT     M36  ; Left    Safety  Door    Down
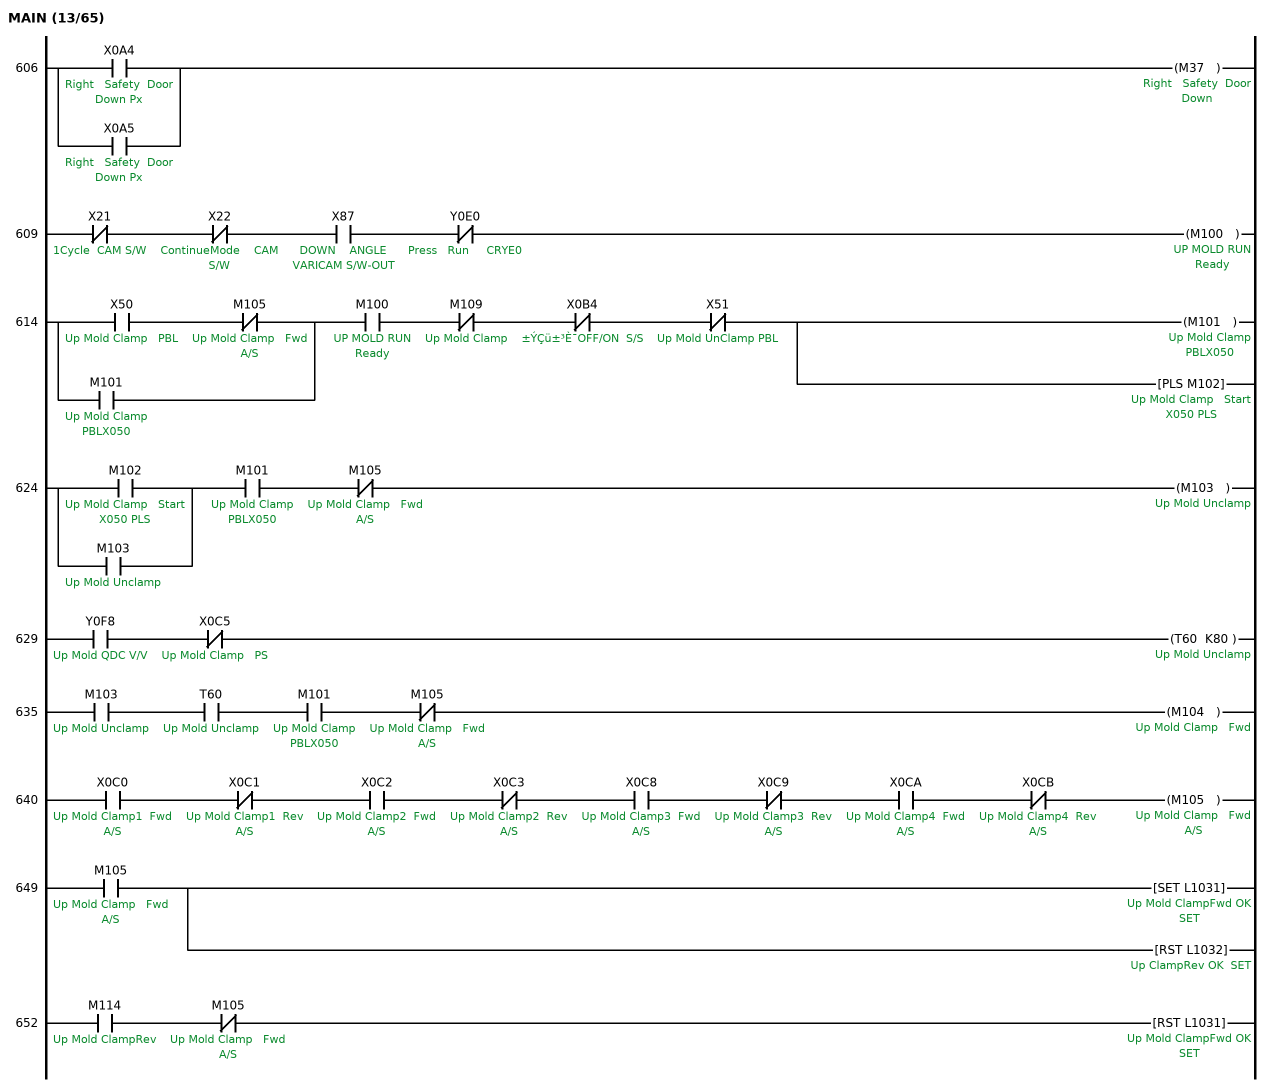
606   LD      X0A4  ; Right   Safety  Door    Down Px
      OR      X0A5  ; Right   Safety  Door    Down Px
      OUT     M37  ; Right   Safety  Door    Down
609   LDI     X21  ; 1Cycle  CAM S/W
      ANI     X22  ; ContinueMode    CAM S/W
      AND     X87  ; DOWN    ANGLE   VARICAM S/W-OUT
      ANI     Y0E0  ; Press   Run     CRYE0
      OUT     M100  ; UP MOLD RUN     Ready
614   LD      X50  ; Up Mold Clamp   PBL
      ANI     M105  ; Up Mold Clamp   Fwd A/S
      OR      M101  ; Up Mold Clamp   PBLX050
      AND     M100  ; UP MOLD RUN     Ready
      ANI     M109  ; Up Mold Clamp
      ANI     X0B4  ; ±ÝÇü±³È¯OFF/ON  S/S
      ANI     X51  ; Up Mold UnClamp PBL
      OUT     M101  ; Up Mold Clamp   PBLX050
      PLS     M102  ; Up Mold Clamp   Start   X050 PLS
624   LD      M102  ; Up Mold Clamp   Start   X050 PLS
      OR      M103  ; Up Mold Unclamp
      AND     M101  ; Up Mold Clamp   PBLX050
      ANI     M105  ; Up Mold Clamp   Fwd A/S
      OUT     M103  ; Up Mold Unclamp
629   LD      Y0F8  ; Up Mold QDC V/V
      ANI     X0C5  ; Up Mold Clamp   PS
      OUT     T60 K80  ; Up Mold Unclamp
635   LD      M103  ; Up Mold Unclamp
      AND     T60  ; Up Mold Unclamp
      AND     M101  ; Up Mold Clamp   PBLX050
      ANI     M105  ; Up Mold Clamp   Fwd A/S
      OUT     M104  ; Up Mold Clamp   Fwd
640   LD      X0C0  ; Up Mold Clamp1  Fwd A/S
      ANI     X0C1  ; Up Mold Clamp1  Rev A/S
      AND     X0C2  ; Up Mold Clamp2  Fwd A/S
      ANI     X0C3  ; Up Mold Clamp2  Rev A/S
      AND     X0C8  ; Up Mold Clamp3  Fwd A/S
      ANI     X0C9  ; Up Mold Clamp3  Rev A/S
      AND     X0CA  ; Up Mold Clamp4  Fwd A/S
      ANI     X0CB  ; Up Mold Clamp4  Rev A/S
      OUT     M105  ; Up Mold Clamp   Fwd A/S
649   LD      M105  ; Up Mold Clamp   Fwd A/S
      SET     L1031  ; Up Mold ClampFwd OK  SET
      RST     L1032  ; Up ClampRev OK  SET
652   LD      M114  ; Up Mold ClampRev
      ANI     M105  ; Up Mold Clamp   Fwd A/S
      RST     L1031  ; Up Mold ClampFwd OK  SET
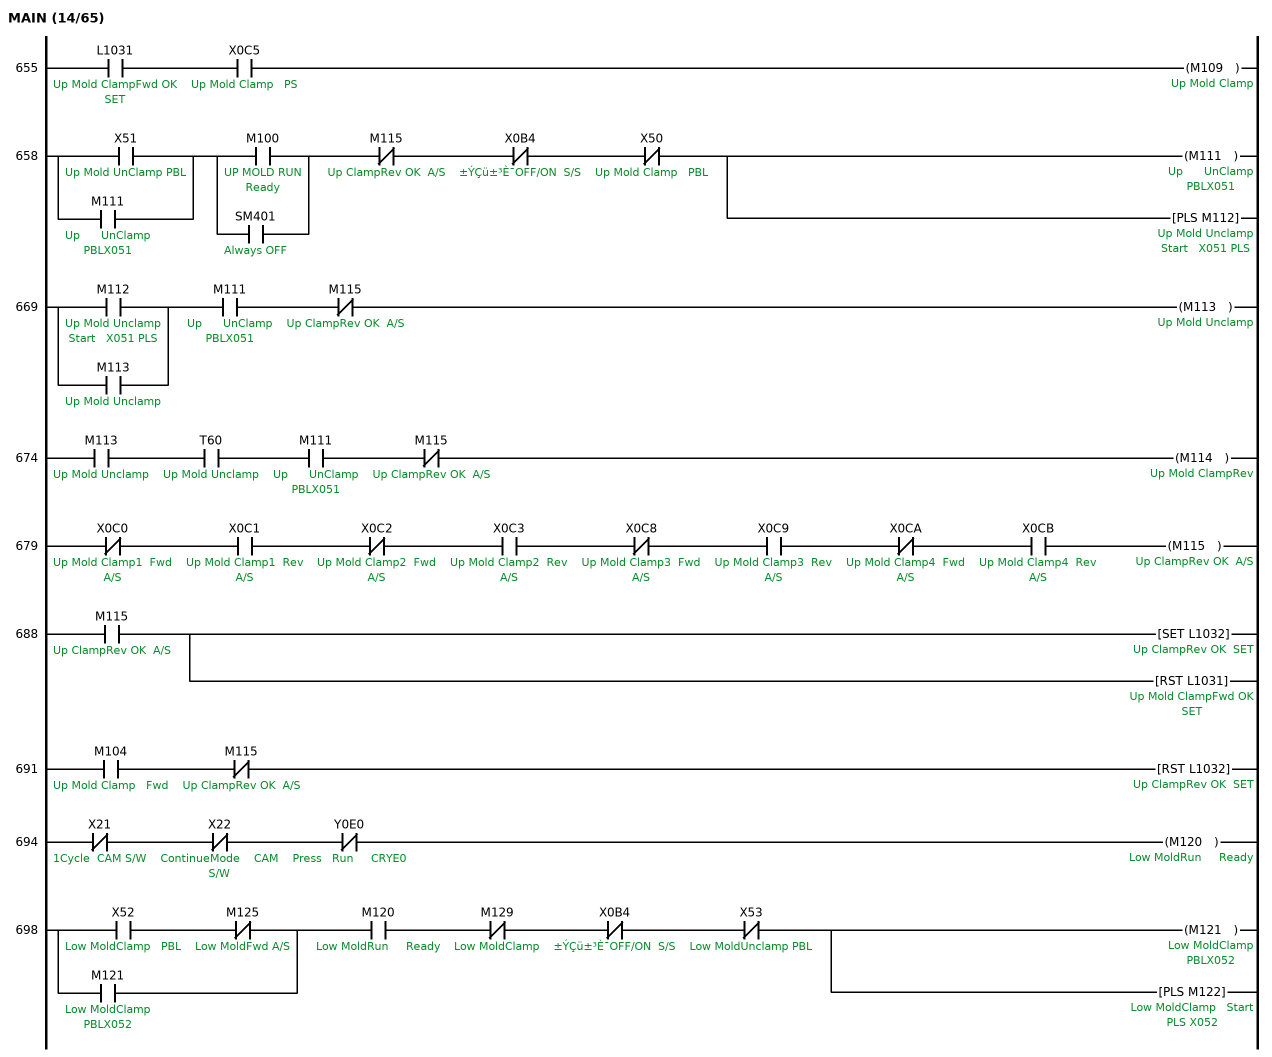
655   LD      L1031  ; Up Mold ClampFwd OK  SET
      AND     X0C5  ; Up Mold Clamp   PS
      OUT     M109  ; Up Mold Clamp
658   LD      X51  ; Up Mold UnClamp PBL
      OR      M111  ; Up      UnClamp PBLX051
      LD      M100  ; UP MOLD RUN     Ready
      OR      SM401  ; Always OFF
      ANB
      ANI     M115  ; Up ClampRev OK  A/S
      ANI     X0B4  ; ±ÝÇü±³È¯OFF/ON  S/S
      ANI     X50  ; Up Mold Clamp   PBL
      OUT     M111  ; Up      UnClamp PBLX051
      PLS     M112  ; Up Mold Unclamp Start   X051 PLS
669   LD      M112  ; Up Mold Unclamp Start   X051 PLS
      OR      M113  ; Up Mold Unclamp
      AND     M111  ; Up      UnClamp PBLX051
      ANI     M115  ; Up ClampRev OK  A/S
      OUT     M113  ; Up Mold Unclamp
674   LD      M113  ; Up Mold Unclamp
      AND     T60  ; Up Mold Unclamp
      AND     M111  ; Up      UnClamp PBLX051
      ANI     M115  ; Up ClampRev OK  A/S
      OUT     M114  ; Up Mold ClampRev
679   LDI     X0C0  ; Up Mold Clamp1  Fwd A/S
      AND     X0C1  ; Up Mold Clamp1  Rev A/S
      ANI     X0C2  ; Up Mold Clamp2  Fwd A/S
      AND     X0C3  ; Up Mold Clamp2  Rev A/S
      ANI     X0C8  ; Up Mold Clamp3  Fwd A/S
      AND     X0C9  ; Up Mold Clamp3  Rev A/S
      ANI     X0CA  ; Up Mold Clamp4  Fwd A/S
      AND     X0CB  ; Up Mold Clamp4  Rev A/S
      OUT     M115  ; Up ClampRev OK  A/S
688   LD      M115  ; Up ClampRev OK  A/S
      SET     L1032  ; Up ClampRev OK  SET
      RST     L1031  ; Up Mold ClampFwd OK  SET
691   LD      M104  ; Up Mold Clamp   Fwd
      ANI     M115  ; Up ClampRev OK  A/S
      RST     L1032  ; Up ClampRev OK  SET
694   LDI     X21  ; 1Cycle  CAM S/W
      ANI     X22  ; ContinueMode    CAM S/W
      ANI     Y0E0  ; Press   Run     CRYE0
      OUT     M120  ; Low MoldRun     Ready
698   LD      X52  ; Low MoldClamp   PBL
      ANI     M125  ; Low MoldFwd A/S
      OR      M121  ; Low MoldClamp   PBLX052
      AND     M120  ; Low MoldRun     Ready
      ANI     M129  ; Low MoldClamp
      ANI     X0B4  ; ±ÝÇü±³È¯OFF/ON  S/S
      ANI     X53  ; Low MoldUnclamp PBL
      OUT     M121  ; Low MoldClamp   PBLX052
      PLS     M122  ; Low MoldClamp   Start   PLS X052
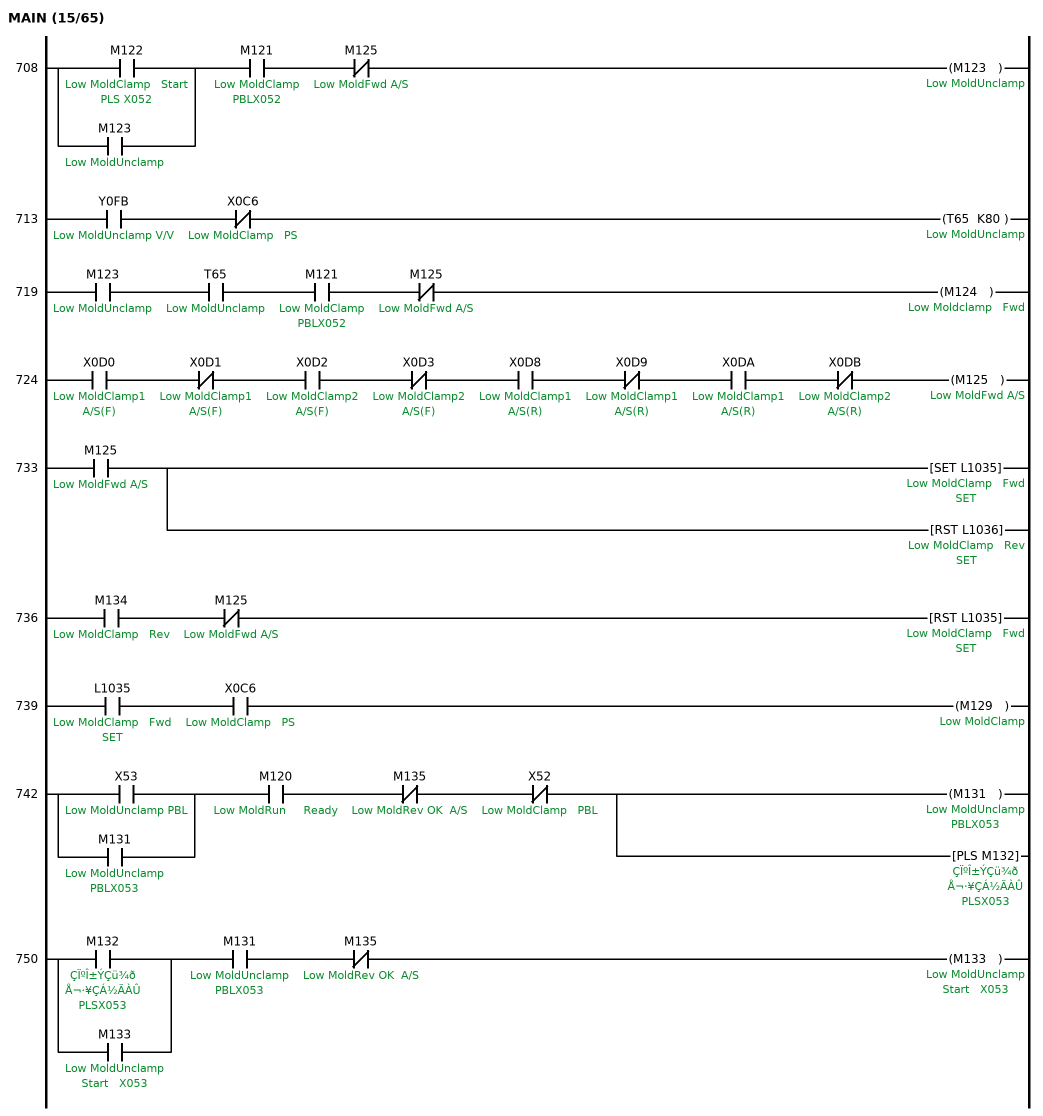
708   LD      M122  ; Low MoldClamp   Start   PLS X052
      OR      M123  ; Low MoldUnclamp
      AND     M121  ; Low MoldClamp   PBLX052
      ANI     M125  ; Low MoldFwd A/S
      OUT     M123  ; Low MoldUnclamp
713   LD      Y0FB  ; Low MoldUnclamp V/V
      ANI     X0C6  ; Low MoldClamp   PS
      OUT     T65 K80  ; Low MoldUnclamp
719   LD      M123  ; Low MoldUnclamp
      AND     T65  ; Low MoldUnclamp
      AND     M121  ; Low MoldClamp   PBLX052
      ANI     M125  ; Low MoldFwd A/S
      OUT     M124  ; Low Moldclamp   Fwd
724   LD      X0D0  ; Low MoldClamp1  A/S(F)
      ANI     X0D1  ; Low MoldClamp1  A/S(F)
      AND     X0D2  ; Low MoldClamp2  A/S(F)
      ANI     X0D3  ; Low MoldClamp2  A/S(F)
      AND     X0D8  ; Low MoldClamp1  A/S(R)
      ANI     X0D9  ; Low MoldClamp1  A/S(R)
      AND     X0DA  ; Low MoldClamp1  A/S(R)
      ANI     X0DB  ; Low MoldClamp2  A/S(R)
      OUT     M125  ; Low MoldFwd A/S
733   LD      M125  ; Low MoldFwd A/S
      SET     L1035  ; Low MoldClamp   Fwd SET
      RST     L1036  ; Low MoldClamp   Rev SET
736   LD      M134  ; Low MoldClamp   Rev
      ANI     M125  ; Low MoldFwd A/S
      RST     L1035  ; Low MoldClamp   Fwd SET
739   LD      L1035  ; Low MoldClamp   Fwd SET
      AND     X0C6  ; Low MoldClamp   PS
      OUT     M129  ; Low MoldClamp
742   LD      X53  ; Low MoldUnclamp PBL
      OR      M131  ; Low MoldUnclamp PBLX053
      AND     M120  ; Low MoldRun     Ready
      ANI     M135  ; Low MoldRev OK  A/S
      ANI     X52  ; Low MoldClamp   PBL
      OUT     M131  ; Low MoldUnclamp PBLX053
      PLS     M132  ; ÇÏºÎ±ÝÇü¾ðÅ¬·¥ÇÁ½ÃÀÛ    PLSX053
750   LD      M132  ; ÇÏºÎ±ÝÇü¾ðÅ¬·¥ÇÁ½ÃÀÛ    PLSX053
      OR      M133  ; Low MoldUnclamp Start   X053
      AND     M131  ; Low MoldUnclamp PBLX053
      ANI     M135  ; Low MoldRev OK  A/S
      OUT     M133  ; Low MoldUnclamp Start   X053
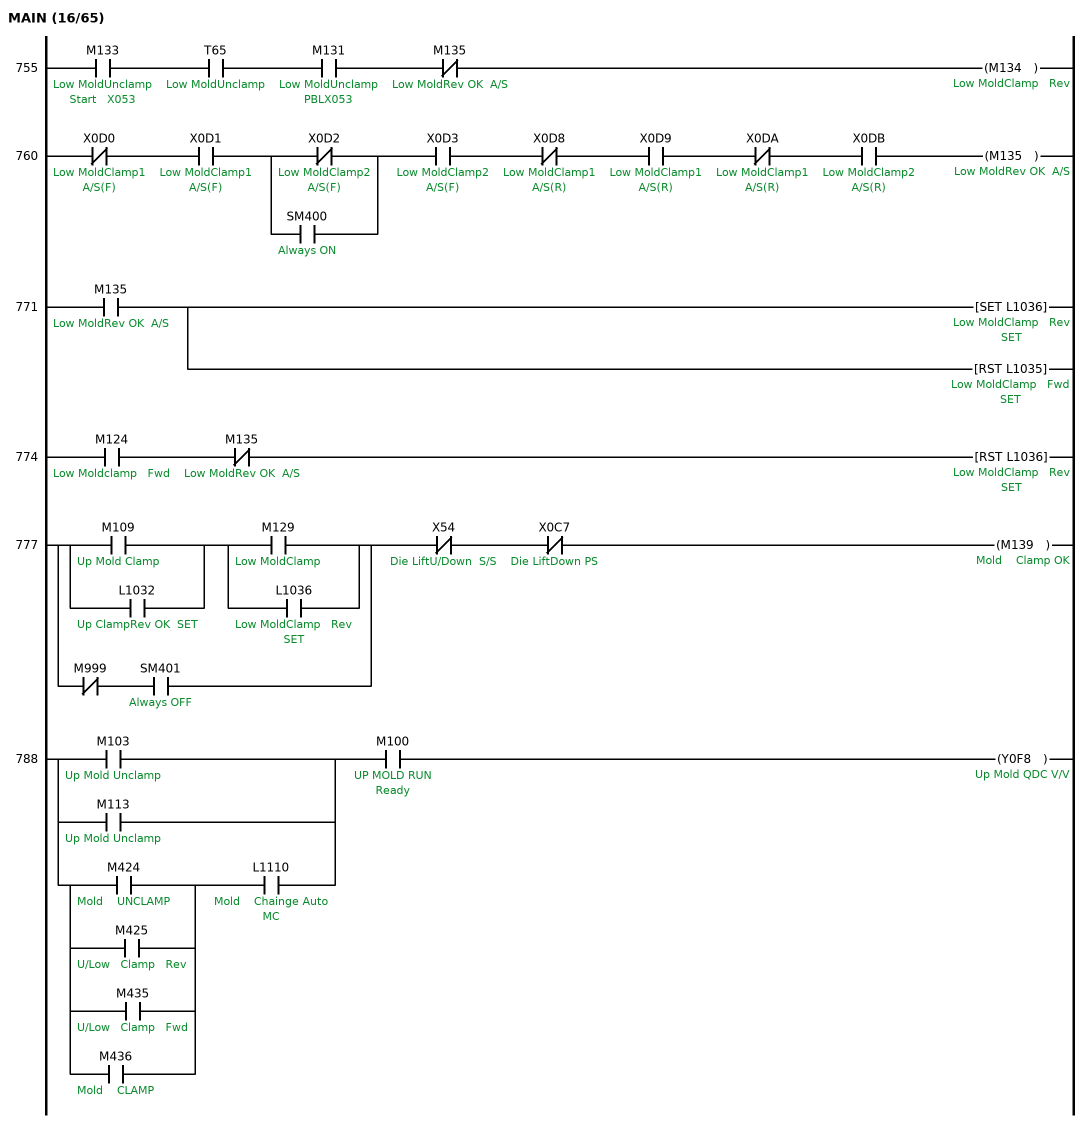
755   LD      M133  ; Low MoldUnclamp Start   X053
      AND     T65  ; Low MoldUnclamp
      AND     M131  ; Low MoldUnclamp PBLX053
      ANI     M135  ; Low MoldRev OK  A/S
      OUT     M134  ; Low MoldClamp   Rev
760   LDI     X0D0  ; Low MoldClamp1  A/S(F)
      AND     X0D1  ; Low MoldClamp1  A/S(F)
      LDI     X0D2  ; Low MoldClamp2  A/S(F)
      OR      SM400  ; Always ON
      ANB
      AND     X0D3  ; Low MoldClamp2  A/S(F)
      ANI     X0D8  ; Low MoldClamp1  A/S(R)
      AND     X0D9  ; Low MoldClamp1  A/S(R)
      ANI     X0DA  ; Low MoldClamp1  A/S(R)
      AND     X0DB  ; Low MoldClamp2  A/S(R)
      OUT     M135  ; Low MoldRev OK  A/S
771   LD      M135  ; Low MoldRev OK  A/S
      SET     L1036  ; Low MoldClamp   Rev SET
      RST     L1035  ; Low MoldClamp   Fwd SET
774   LD      M124  ; Low Moldclamp   Fwd
      ANI     M135  ; Low MoldRev OK  A/S
      RST     L1036  ; Low MoldClamp   Rev SET
777   LD      M109  ; Up Mold Clamp
      OR      L1032  ; Up ClampRev OK  SET
      LD      M129  ; Low MoldClamp
      OR      L1036  ; Low MoldClamp   Rev SET
      ANB
      LDI     M999
      AND     SM401  ; Always OFF
      ORB
      ANI     X54  ; Die LiftU/Down  S/S
      ANI     X0C7  ; Die LiftDown PS
      OUT     M139  ; Mold    Clamp OK
788   LD      M103  ; Up Mold Unclamp
      OR      M113  ; Up Mold Unclamp
      LD      M424  ; Mold    UNCLAMP
      OR      M425  ; U/Low   Clamp   Rev
      OR      M435  ; U/Low   Clamp   Fwd
      OR      M436  ; Mold    CLAMP
      AND     L1110  ; Mold    Chainge Auto MC
      ORB
      AND     M100  ; UP MOLD RUN     Ready
      OUT     Y0F8  ; Up Mold QDC V/V
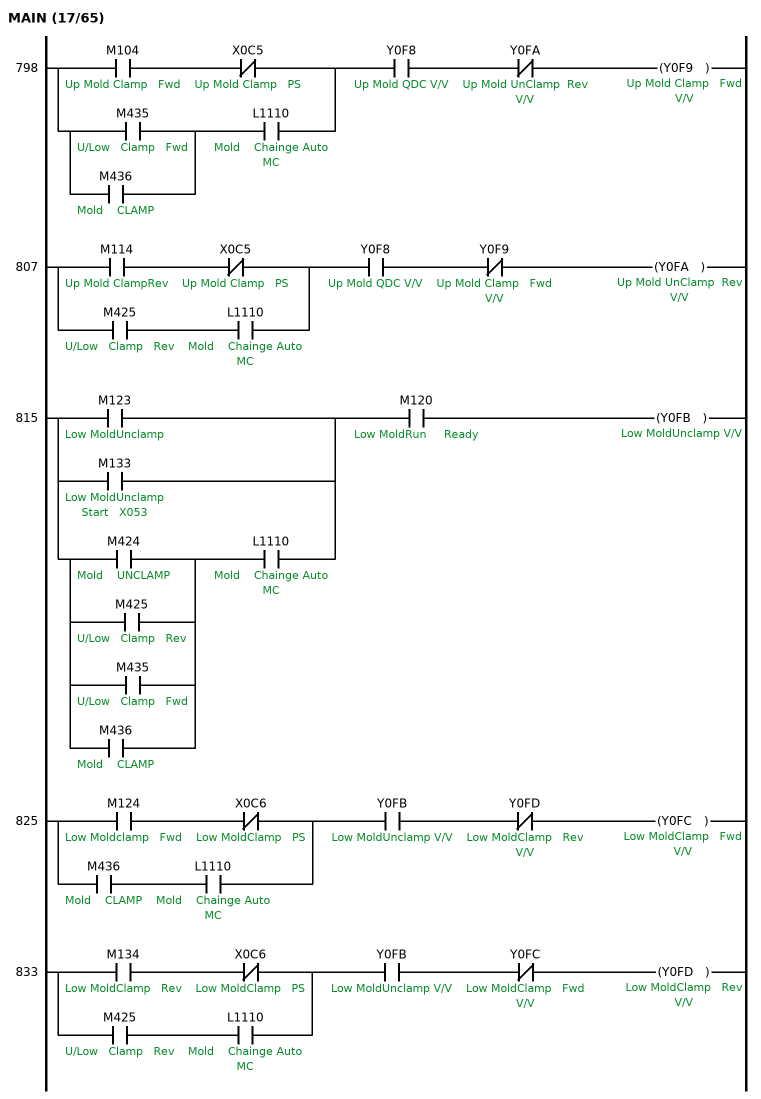
798   LD      M104  ; Up Mold Clamp   Fwd
      ANI     X0C5  ; Up Mold Clamp   PS
      LD      M435  ; U/Low   Clamp   Fwd
      OR      M436  ; Mold    CLAMP
      AND     L1110  ; Mold    Chainge Auto MC
      ORB
      AND     Y0F8  ; Up Mold QDC V/V
      ANI     Y0FA  ; Up Mold UnClamp  Rev V/V
      OUT     Y0F9  ; Up Mold Clamp   Fwd V/V
807   LD      M114  ; Up Mold ClampRev
      ANI     X0C5  ; Up Mold Clamp   PS
      LD      M425  ; U/Low   Clamp   Rev
      AND     L1110  ; Mold    Chainge Auto MC
      ORB
      AND     Y0F8  ; Up Mold QDC V/V
      ANI     Y0F9  ; Up Mold Clamp   Fwd V/V
      OUT     Y0FA  ; Up Mold UnClamp  Rev V/V
815   LD      M123  ; Low MoldUnclamp
      OR      M133  ; Low MoldUnclamp Start   X053
      LD      M424  ; Mold    UNCLAMP
      OR      M425  ; U/Low   Clamp   Rev
      OR      M435  ; U/Low   Clamp   Fwd
      OR      M436  ; Mold    CLAMP
      AND     L1110  ; Mold    Chainge Auto MC
      ORB
      AND     M120  ; Low MoldRun     Ready
      OUT     Y0FB  ; Low MoldUnclamp V/V
825   LD      M124  ; Low Moldclamp   Fwd
      ANI     X0C6  ; Low MoldClamp   PS
      LD      M436  ; Mold    CLAMP
      AND     L1110  ; Mold    Chainge Auto MC
      ORB
      AND     Y0FB  ; Low MoldUnclamp V/V
      ANI     Y0FD  ; Low MoldClamp   Rev V/V
      OUT     Y0FC  ; Low MoldClamp   Fwd V/V
833   LD      M134  ; Low MoldClamp   Rev
      ANI     X0C6  ; Low MoldClamp   PS
      LD      M425  ; U/Low   Clamp   Rev
      AND     L1110  ; Mold    Chainge Auto MC
      ORB
      AND     Y0FB  ; Low MoldUnclamp V/V
      ANI     Y0FC  ; Low MoldClamp   Fwd V/V
      OUT     Y0FD  ; Low MoldClamp   Rev V/V
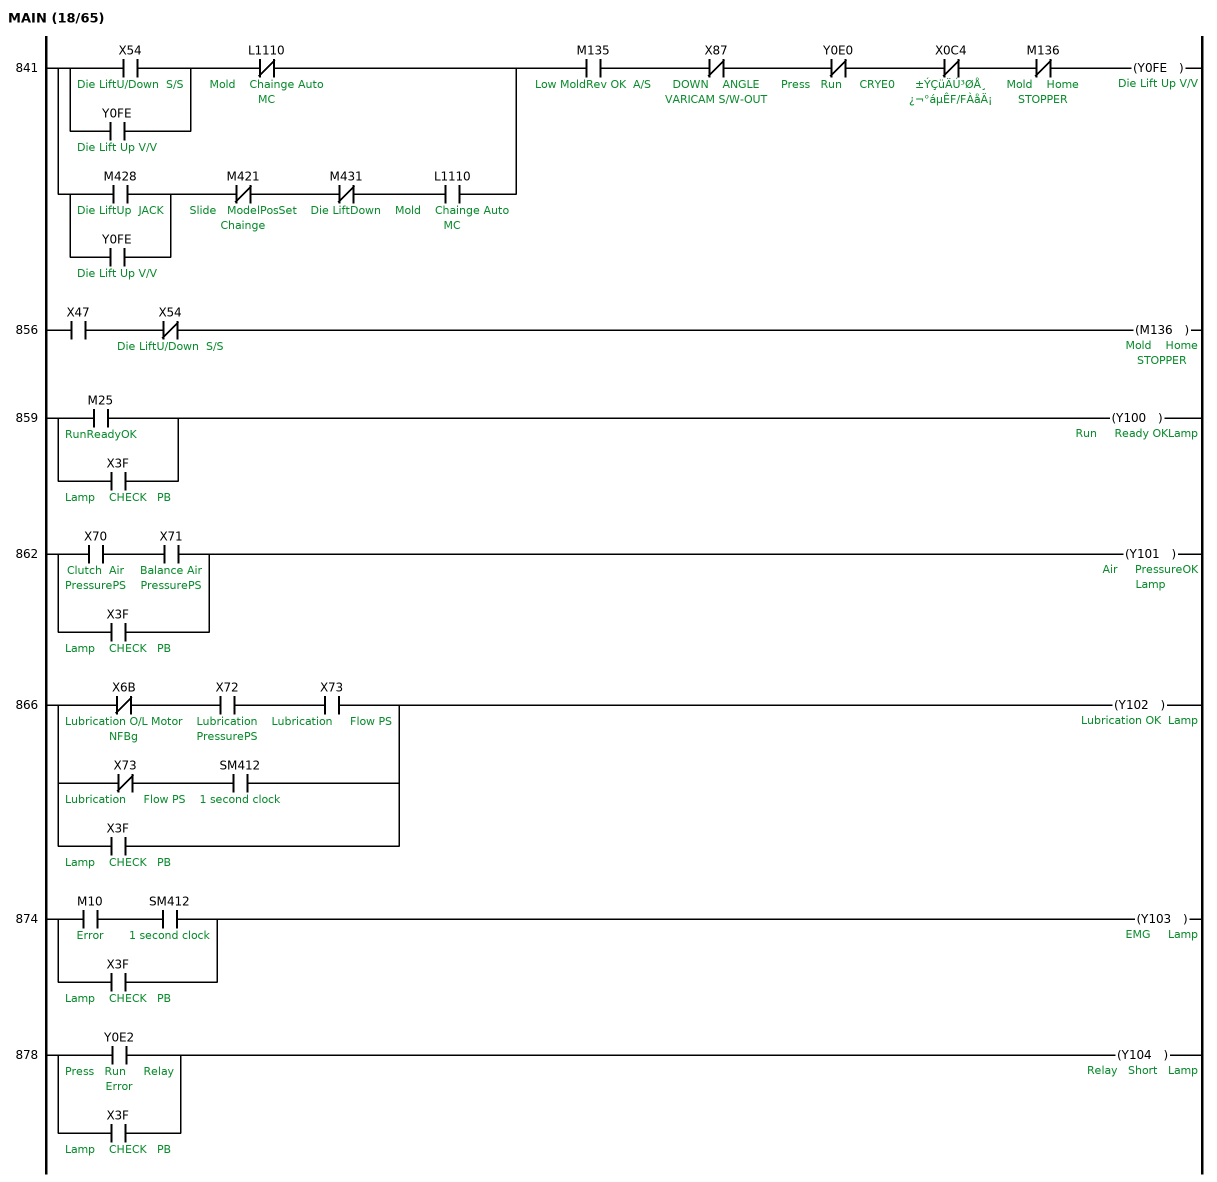
841   LD      X54  ; Die LiftU/Down  S/S
      OR      Y0FE  ; Die Lift Up V/V
      ANI     L1110  ; Mold    Chainge Auto MC
      LD      M428  ; Die LiftUp  JACK
      OR      Y0FE  ; Die Lift Up V/V
      ANI     M421  ; Slide   ModelPosSet     Chainge
      ANI     M431  ; Die LiftDown
      AND     L1110  ; Mold    Chainge Auto MC
      ORB
      AND     M135  ; Low MoldRev OK  A/S
      ANI     X87  ; DOWN    ANGLE   VARICAM S/W-OUT
      ANI     Y0E0  ; Press   Run     CRYE0
      ANI     X0C4  ; ±ÝÇüÄÚ³ØÅ¸ ¿¬°áµÊF/FÀåÄ¡
      ANI     M136  ; Mold    Home    STOPPER
      OUT     Y0FE  ; Die Lift Up V/V
856   LD      X47
      ANI     X54  ; Die LiftU/Down  S/S
      OUT     M136  ; Mold    Home    STOPPER
859   LD      M25  ; RunReadyOK
      OR      X3F  ; Lamp    CHECK   PB
      OUT     Y100  ; Run     Ready OKLamp
862   LD      X70  ; Clutch  Air     PressurePS
      AND     X71  ; Balance Air     PressurePS
      OR      X3F  ; Lamp    CHECK   PB
      OUT     Y101  ; Air     PressureOK Lamp
866   LDI     X6B  ; Lubrication O/L Motor   NFBg
      AND     X72  ; Lubrication     PressurePS
      AND     X73  ; Lubrication     Flow PS
      LDI     X73  ; Lubrication     Flow PS
      AND     SM412  ; 1 second clock
      ORB
      OR      X3F  ; Lamp    CHECK   PB
      OUT     Y102  ; Lubrication OK  Lamp
874   LD      M10  ; Error
      AND     SM412  ; 1 second clock
      OR      X3F  ; Lamp    CHECK   PB
      OUT     Y103  ; EMG     Lamp
878   LD      Y0E2  ; Press   Run     Relay   Error
      OR      X3F  ; Lamp    CHECK   PB
      OUT     Y104  ; Relay   Short   Lamp
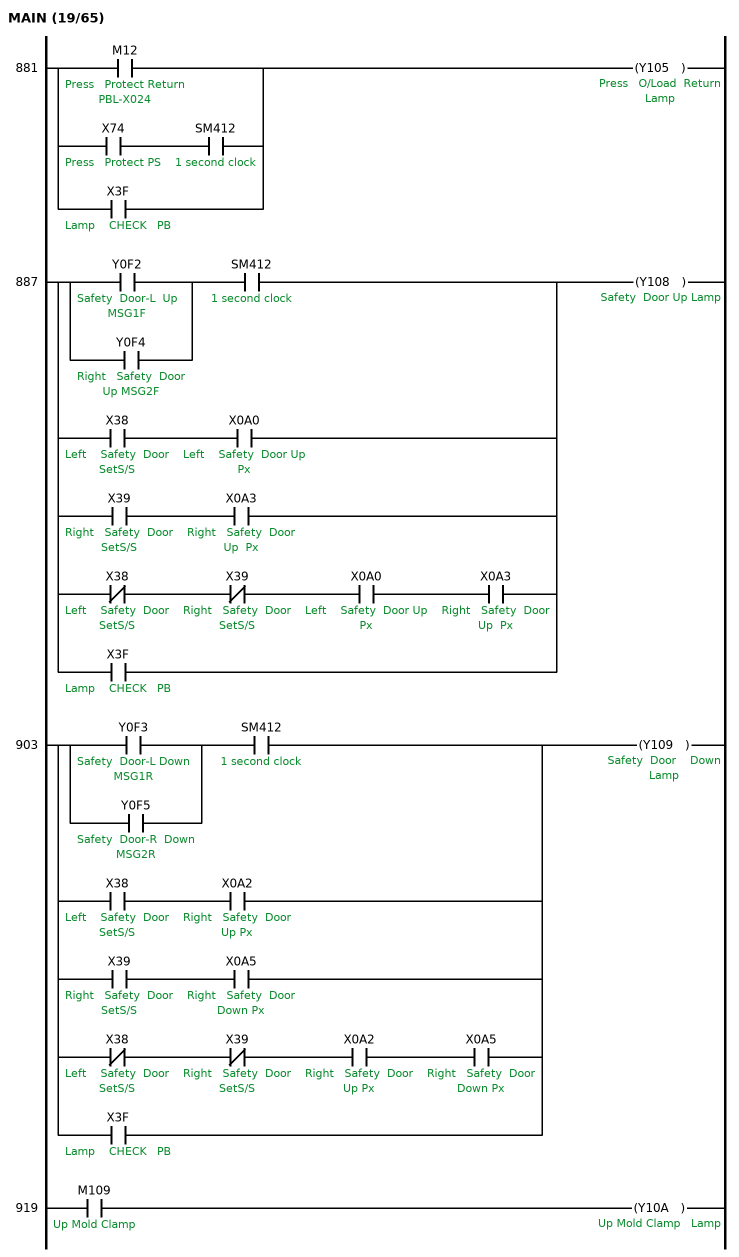
881   LD      M12  ; Press   Protect Return  PBL-X024
      LD      X74  ; Press   Protect PS
      AND     SM412  ; 1 second clock
      ORB
      OR      X3F  ; Lamp    CHECK   PB
      OUT     Y105  ; Press   O/Load  Return  Lamp
887   LD      Y0F2  ; Safety  Door-L  Up MSG1F
      OR      Y0F4  ; Right   Safety  Door Up MSG2F
      AND     SM412  ; 1 second clock
      LD      X38  ; Left    Safety  Door SetS/S
      AND     X0A0  ; Left    Safety  Door Up Px
      ORB
      LD      X39  ; Right   Safety  Door SetS/S
      AND     X0A3  ; Right   Safety  Door Up  Px
      ORB
      LDI     X38  ; Left    Safety  Door SetS/S
      ANI     X39  ; Right   Safety  Door SetS/S
      AND     X0A0  ; Left    Safety  Door Up Px
      AND     X0A3  ; Right   Safety  Door Up  Px
      ORB
      OR      X3F  ; Lamp    CHECK   PB
      OUT     Y108  ; Safety  Door Up Lamp
903   LD      Y0F3  ; Safety  Door-L Down     MSG1R
      OR      Y0F5  ; Safety  Door-R  Down    MSG2R
      AND     SM412  ; 1 second clock
      LD      X38  ; Left    Safety  Door SetS/S
      AND     X0A2  ; Right   Safety  Door Up Px
      ORB
      LD      X39  ; Right   Safety  Door SetS/S
      AND     X0A5  ; Right   Safety  Door    Down Px
      ORB
      LDI     X38  ; Left    Safety  Door SetS/S
      ANI     X39  ; Right   Safety  Door SetS/S
      AND     X0A2  ; Right   Safety  Door Up Px
      AND     X0A5  ; Right   Safety  Door    Down Px
      ORB
      OR      X3F  ; Lamp    CHECK   PB
      OUT     Y109  ; Safety  Door    Down    Lamp
919   LD      M109  ; Up Mold Clamp
      OUT     Y10A  ; Up Mold Clamp   Lamp
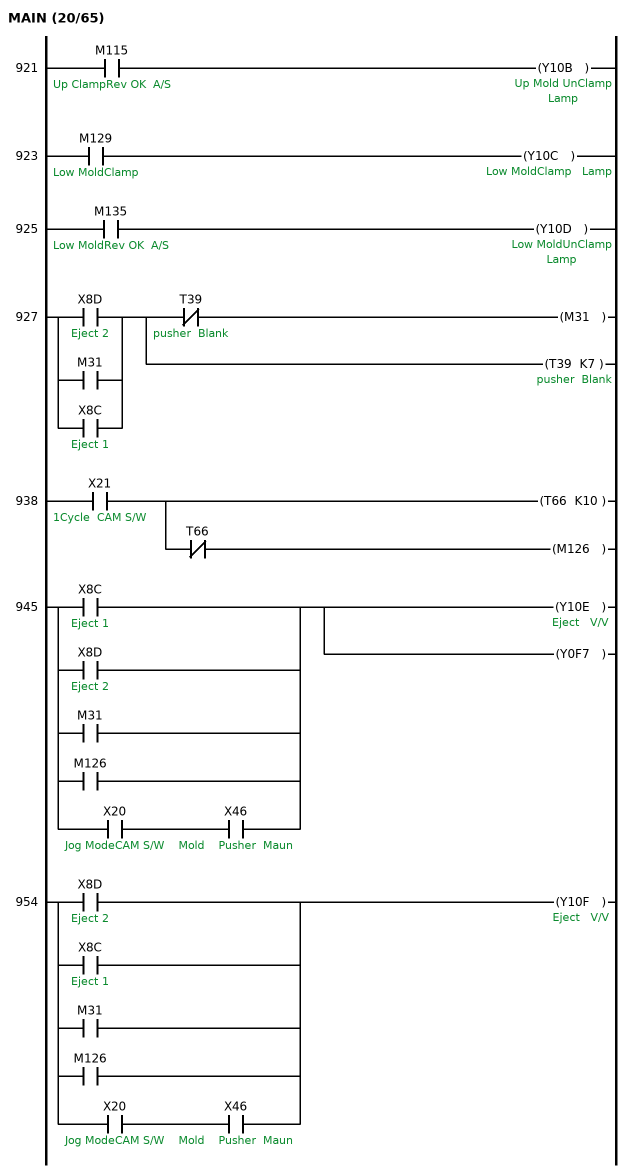
921   LD      M115  ; Up ClampRev OK  A/S
      OUT     Y10B  ; Up Mold UnClamp Lamp
923   LD      M129  ; Low MoldClamp
      OUT     Y10C  ; Low MoldClamp   Lamp
925   LD      M135  ; Low MoldRev OK  A/S
      OUT     Y10D  ; Low MoldUnClamp Lamp
927   LD      X8D  ; Eject 2
      OR      M31
      OR      X8C  ; Eject 1
      MPS
      ANI     T39  ; pusher  Blank
      OUT     M31
      MPP
      OUT     T39 K7  ; pusher  Blank
938   LD      X21  ; 1Cycle  CAM S/W
      OUT     T66 K10
      ANI     T66
      OUT     M126
945   LD      X8C  ; Eject 1
      OR      X8D  ; Eject 2
      OR      M31
      OR      M126
      LD      X20  ; Jog ModeCAM S/W
      AND     X46  ; Mold    Pusher  Maun
      ORB
      OUT     Y10E  ; Eject   V/V
      OUT     Y0F7
954   LD      X8D  ; Eject 2
      OR      X8C  ; Eject 1
      OR      M31
      OR      M126
      LD      X20  ; Jog ModeCAM S/W
      AND     X46  ; Mold    Pusher  Maun
      ORB
      OUT     Y10F  ; Eject   V/V
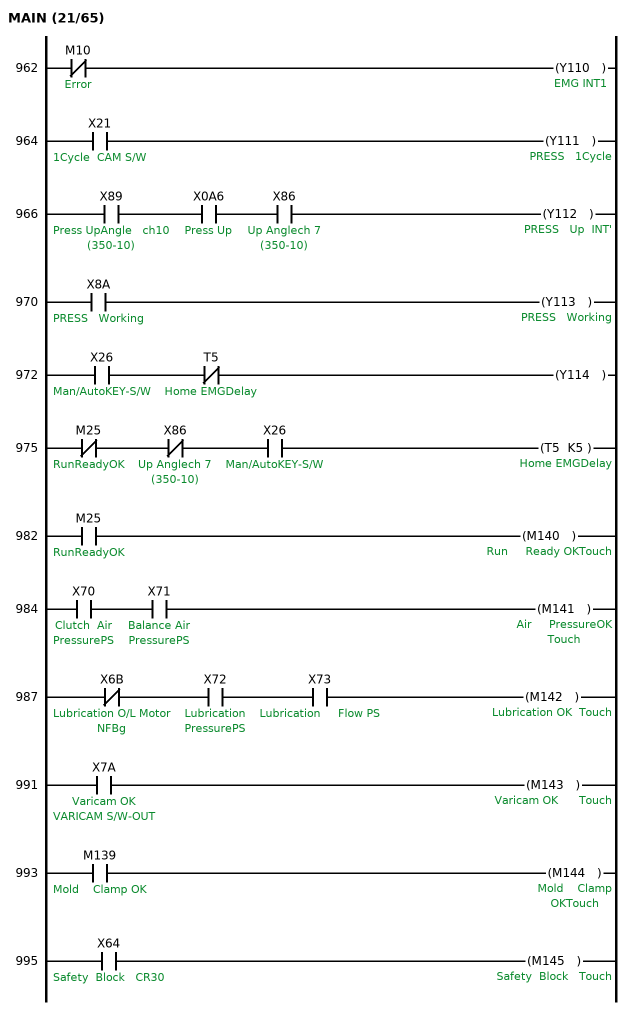
962   LDI     M10  ; Error
      OUT     Y110  ; EMG INT1
964   LD      X21  ; 1Cycle  CAM S/W
      OUT     Y111  ; PRESS   1Cycle
966   LD      X89  ; Press UpAngle   ch10 (350-10)
      AND     X0A6  ; Press Up
      AND     X86  ; Up Anglech 7    (350-10)
      OUT     Y112  ; PRESS   Up  INT'
970   LD      X8A  ; PRESS   Working
      OUT     Y113  ; PRESS   Working
972   LD      X26  ; Man/AutoKEY-S/W
      ANI     T5  ; Home EMGDelay
      OUT     Y114
975   LDI     M25  ; RunReadyOK
      ANI     X86  ; Up Anglech 7    (350-10)
      AND     X26  ; Man/AutoKEY-S/W
      OUT     T5 K5  ; Home EMGDelay
982   LD      M25  ; RunReadyOK
      OUT     M140  ; Run     Ready OKTouch
984   LD      X70  ; Clutch  Air     PressurePS
      AND     X71  ; Balance Air     PressurePS
      OUT     M141  ; Air     PressureOK Touch
987   LDI     X6B  ; Lubrication O/L Motor   NFBg
      AND     X72  ; Lubrication     PressurePS
      AND     X73  ; Lubrication     Flow PS
      OUT     M142  ; Lubrication OK  Touch
991   LD      X7A  ; Varicam OK      VARICAM S/W-OUT
      OUT     M143  ; Varicam OK      Touch
993   LD      M139  ; Mold    Clamp OK
      OUT     M144  ; Mold    Clamp OKTouch
995   LD      X64  ; Safety  Block   CR30
      OUT     M145  ; Safety  Block   Touch
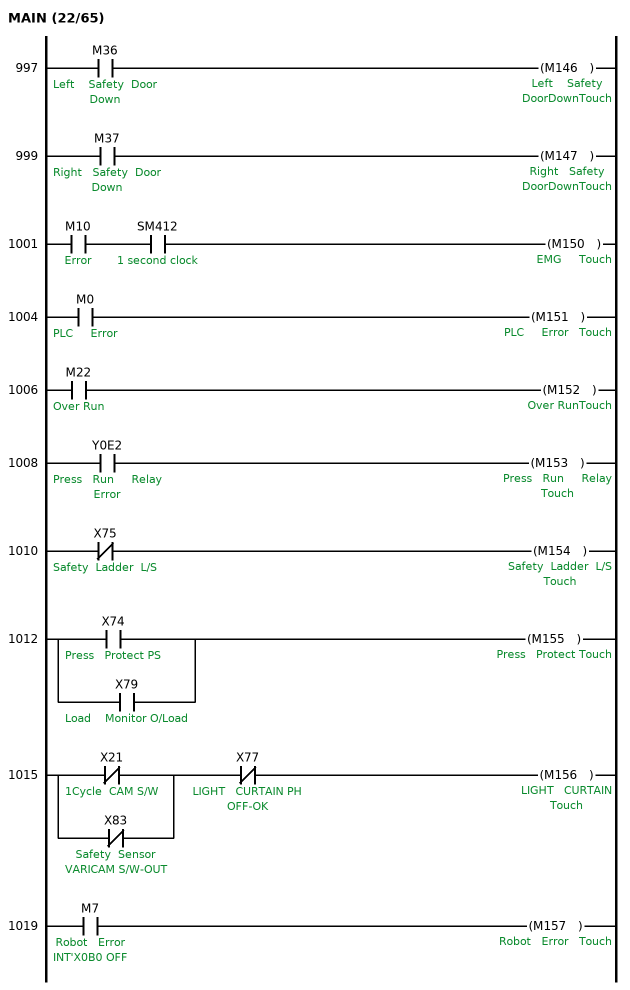
997   LD      M36  ; Left    Safety  Door    Down
      OUT     M146  ; Left    Safety  DoorDownTouch
999   LD      M37  ; Right   Safety  Door    Down
      OUT     M147  ; Right   Safety  DoorDownTouch
1001  LD      M10  ; Error
      AND     SM412  ; 1 second clock
      OUT     M150  ; EMG     Touch
1004  LD      M0  ; PLC     Error
      OUT     M151  ; PLC     Error   Touch
1006  LD      M22  ; Over Run
      OUT     M152  ; Over RunTouch
1008  LD      Y0E2  ; Press   Run     Relay   Error
      OUT     M153  ; Press   Run     Relay   Touch
1010  LDI     X75  ; Safety  Ladder  L/S
      OUT     M154  ; Safety  Ladder  L/S     Touch
1012  LD      X74  ; Press   Protect PS
      OR      X79  ; Load    Monitor O/Load
      OUT     M155  ; Press   Protect Touch
1015  LDI     X21  ; 1Cycle  CAM S/W
      ORI     X83  ; Safety  Sensor  VARICAM S/W-OUT
      ANI     X77  ; LIGHT   CURTAIN PH      OFF-OK
      OUT     M156  ; LIGHT   CURTAIN Touch
1019  LD      M7  ; Robot   Error   INT'X0B0 OFF
      OUT     M157  ; Robot   Error   Touch
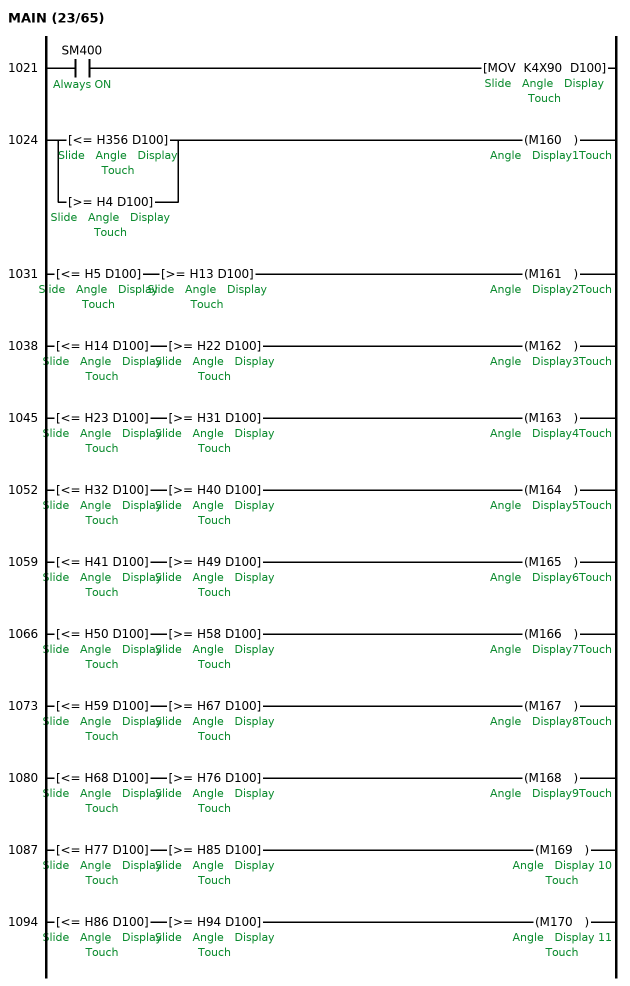
1021  LD      SM400  ; Always ON
      MOV     K4X90 D100  ; Slide   Angle   In / Slide   Angle   Display Touch
1024  LD<=    H356 D100  ; Slide   Angle   Display Touch
      OR>=    H4 D100  ; Slide   Angle   Display Touch
      OUT     M160  ; Angle   Display1Touch
1031  LD<=    H5 D100  ; Slide   Angle   Display Touch
      AND>=   H13 D100  ; Slide   Angle   Display Touch
      OUT     M161  ; Angle   Display2Touch
1038  LD<=    H14 D100  ; Slide   Angle   Display Touch
      AND>=   H22 D100  ; Slide   Angle   Display Touch
      OUT     M162  ; Angle   Display3Touch
1045  LD<=    H23 D100  ; Slide   Angle   Display Touch
      AND>=   H31 D100  ; Slide   Angle   Display Touch
      OUT     M163  ; Angle   Display4Touch
1052  LD<=    H32 D100  ; Slide   Angle   Display Touch
      AND>=   H40 D100  ; Slide   Angle   Display Touch
      OUT     M164  ; Angle   Display5Touch
1059  LD<=    H41 D100  ; Slide   Angle   Display Touch
      AND>=   H49 D100  ; Slide   Angle   Display Touch
      OUT     M165  ; Angle   Display6Touch
1066  LD<=    H50 D100  ; Slide   Angle   Display Touch
      AND>=   H58 D100  ; Slide   Angle   Display Touch
      OUT     M166  ; Angle   Display7Touch
1073  LD<=    H59 D100  ; Slide   Angle   Display Touch
      AND>=   H67 D100  ; Slide   Angle   Display Touch
      OUT     M167  ; Angle   Display8Touch
1080  LD<=    H68 D100  ; Slide   Angle   Display Touch
      AND>=   H76 D100  ; Slide   Angle   Display Touch
      OUT     M168  ; Angle   Display9Touch
1087  LD<=    H77 D100  ; Slide   Angle   Display Touch
      AND>=   H85 D100  ; Slide   Angle   Display Touch
      OUT     M169  ; Angle   Display 10 Touch
1094  LD<=    H86 D100  ; Slide   Angle   Display Touch
      AND>=   H94 D100  ; Slide   Angle   Display Touch
      OUT     M170  ; Angle   Display 11      Touch
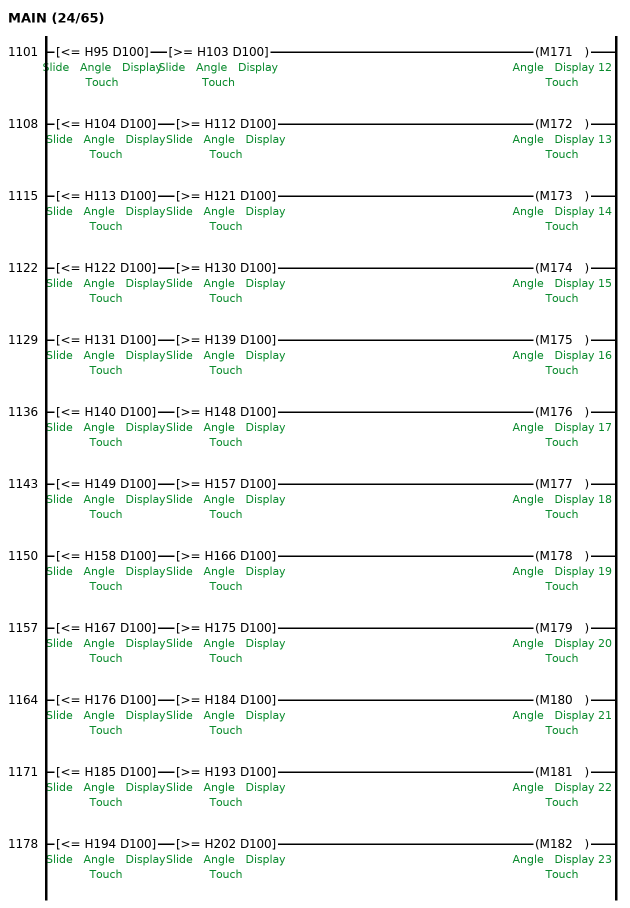
1101  LD<=    H95 D100  ; Slide   Angle   Display Touch
      AND>=   H103 D100  ; Slide   Angle   Display Touch
      OUT     M171  ; Angle   Display 12      Touch
1108  LD<=    H104 D100  ; Slide   Angle   Display Touch
      AND>=   H112 D100  ; Slide   Angle   Display Touch
      OUT     M172  ; Angle   Display 13      Touch
1115  LD<=    H113 D100  ; Slide   Angle   Display Touch
      AND>=   H121 D100  ; Slide   Angle   Display Touch
      OUT     M173  ; Angle   Display 14      Touch
1122  LD<=    H122 D100  ; Slide   Angle   Display Touch
      AND>=   H130 D100  ; Slide   Angle   Display Touch
      OUT     M174  ; Angle   Display 15      Touch
1129  LD<=    H131 D100  ; Slide   Angle   Display Touch
      AND>=   H139 D100  ; Slide   Angle   Display Touch
      OUT     M175  ; Angle   Display 16      Touch
1136  LD<=    H140 D100  ; Slide   Angle   Display Touch
      AND>=   H148 D100  ; Slide   Angle   Display Touch
      OUT     M176  ; Angle   Display 17      Touch
1143  LD<=    H149 D100  ; Slide   Angle   Display Touch
      AND>=   H157 D100  ; Slide   Angle   Display Touch
      OUT     M177  ; Angle   Display 18      Touch
1150  LD<=    H158 D100  ; Slide   Angle   Display Touch
      AND>=   H166 D100  ; Slide   Angle   Display Touch
      OUT     M178  ; Angle   Display 19      Touch
1157  LD<=    H167 D100  ; Slide   Angle   Display Touch
      AND>=   H175 D100  ; Slide   Angle   Display Touch
      OUT     M179  ; Angle   Display 20      Touch
1164  LD<=    H176 D100  ; Slide   Angle   Display Touch
      AND>=   H184 D100  ; Slide   Angle   Display Touch
      OUT     M180  ; Angle   Display 21      Touch
1171  LD<=    H185 D100  ; Slide   Angle   Display Touch
      AND>=   H193 D100  ; Slide   Angle   Display Touch
      OUT     M181  ; Angle   Display 22      Touch
1178  LD<=    H194 D100  ; Slide   Angle   Display Touch
      AND>=   H202 D100  ; Slide   Angle   Display Touch
      OUT     M182  ; Angle   Display 23      Touch
